		(* Fill input data area with method arguments *)
		MEMSET(ADR(aInputData), 0 ,SIZEOF(aInputData));
		nOffset := 0;
		nOffset := nOffset + MEMCPY(ADR(aInputData)+nOffset, ADR(stMoveToBufferData.stInput),	MIN(SIZEOF(stMoveToBufferData.stInput), (SIZEOF(aInputData)-nOffset)) );
		(* Number of input arguments *)
		nNoOfInputArgs := stMoveToBufferData.iNoOfInputArgs;
		(* Set up input argument information *)
		MEMSET(ADR(aInputArgInfo), 0, SIZEOF(aInputArgInfo));
		aInputArgInfo[1].DataType := eUAType_UInt16;
		aInputArgInfo[1].ValueRank := -1;	// -1: Scalar 
		aInputArgInfo[1].nLenData := SIZEOF(stMoveToBufferData.stInput.eInputType);
		aInputArgInfo[2].DataType := eUAType_String;
		aInputArgInfo[2].ValueRank := -1;	// -1: Scalar 
		aInputArgInfo[2].nLenData := SIZEOF(stMoveToBufferData.stInput.sInput);
		aInputArgInfo[3].DataType := eUAType_String;
		aInputArgInfo[3].ValueRank := -1;	// -1: Scalar 
		aInputArgInfo[3].nLenData := SIZEOF(stMoveToBufferData.stInput.sStationID);
		aInputArgInfo[4].DataType := eUAType_UInt16;
		aInputArgInfo[4].ValueRank := -1;	// -1: Scalar 
		aInputArgInfo[4].nLenData := SIZEOF(stMoveToBufferData.stInput.eStationBufferType);
		aInputArgInfo[5].DataType := eUAType_Byte;
		aInputArgInfo[5].ValueRank := -1;	// -1: Scalar 
		aInputArgInfo[5].nLenData := SIZEOF(stMoveToBufferData.stInput.nIndex);
		aInputArgInfo[6].DataType := eUAType_Byte;
		aInputArgInfo[6].ValueRank := -1;	// -1: Scalar 
		aInputArgInfo[6].nLenData := SIZEOF(stMoveToBufferData.stInput.eDirection);
		aInputArgInfo[7].DataType := eUAType_UInt16;
		aInputArgInfo[7].ValueRank := -1;	// -1: Scalar 
		aInputArgInfo[7].nLenData := SIZEOF(stMoveToBufferData.stInput.nFollowID);
		aInputArgInfo[8].DataType := eUAType_Float;
		aInputArgInfo[8].ValueRank := -1;	// -1: Scalar 
		aInputArgInfo[8].nLenData := SIZEOF(stMoveToBufferData.stInput.fVelocity);
		aInputArgInfo[9].DataType := eUAType_Float;
		aInputArgInfo[9].ValueRank := -1;	// -1: Scalar 
		aInputArgInfo[9].nLenData := SIZEOF(stMoveToBufferData.stInput.fAcceleration);
		
		(* Method outputs *)
		(* Clear output data area *)
		(* Number of output arguments *)
		nNoOfOutputArgs := stMoveToBufferData.iNoOfOutputArgs;
		(* Set up output argument information *)
		MEMSET(ADR(aOutputArgInfo), 0, SIZEOF(aOutputArgInfo));
		aOutputArgInfo[1].DataType := eUAType_Uint16;
		aOutputArgInfo[1].ValueRank := -1;
		aOutputArgInfo[1].nLenData := SIZEOF(stMoveToBufferData.stOutput.eStatus);
		aOutputArgInfo[2].DataType := eUAType_String;
		aOutputArgInfo[2].ValueRank := -1;
		aOutputArgInfo[2].nLenData := SIZEOF(stMoveToBufferData.stOutput.sMessage);
		aOutputArgInfo[3].DataType := eUAType_UInt16;
		aOutputArgInfo[3].ValueRank := -1;
		aOutputArgInfo[3].nLenData := SIZEOF(stMoveToBufferData.stOutput.iCommandID);		
		(* Set up output  *)
		MEMSET(ADR(stMoveToBufferData.stOutput), 0, SIZEOF(stMoveToBufferData.stOutput));
		stMoveToBufferData.stOutput.nNumberOfOutputArguments := nNoOfOutputArgs;
		stMoveToBufferData.stOutput.stOutputArgInfo[1] := aOutputArgInfo[1];
		stMoveToBufferData.stOutput.stOutputArgInfo[2] := aOutputArgInfo[2];
		stMoveToBufferData.stOutput.stOutputArgInfo[3] := aOutputArgInfo[3];
	
		(* Execute FB *)
		fbCallMethod.nNumberOfInputArguments := nNoOfInputArgs;
		fbCallMethod.pInputArgInfo := ADR(aInputArgInfo);
		fbCallMethod.cbInputArgInfo := (SIZEOF(aInputArgInfo[1])*nNoOfInputArgs);
		fbCallMethod.pInputArgData := ADR(aInputData);
		fbCallMethod.cbInputArgData := nOffset;
		fbCallMethod.nNumberOfOutputArguments := nNoOfOutputArgs; 
		fbCallMethod.pOutputArgInfo := ADR(aOutputArgInfo); 
		fbCallMethod.cbOutputArgInfo := (SIZEOF(aOutputArgInfo[1]) * nNoOfOutputArgs); 
		fbCallMethod.pOutputArgInfoAndData := ADR(stMoveToBufferData.stOutput);
		fbCallMethod.cbOutputArgInfoAndData := SIZEOF(stMoveToBufferData.stOutput);
		
		stMoveToBufferData.iStatus := 1;
		bCallMethod := TRUE;
		
	ELSIF ( (stMoveToBufferData.iStatus = 1) AND (stMoveToBufferData.stInput.sInput = sInput) ) THEN
		// Method call Completed...
		IF (eStateMethod = E_TrackClientState.Connected) THEN
			// Method call OK
			IF (stMoveToBufferData.stOutput.eStatus = E_MMServerStatus.eMMServerStatus_Success) THEN
				// Method returned OK
				stMoveToBufferData.iStatus := 2;
				iCmdID := stMoveToBufferData.stOutput.iCommandID;
			ELSE
				// Method returned with error
				stMoveToBufferData.iStatus := 3;
				stMoveToBufferData.stOutput.sMessage;
				iCmdID := 0;
			END_IF
		ELSIF (eStateMethod = E_TrackClientState.Error) THEN
			// Method call failed
			stMoveToBufferData.iStatus := 3;
		END_IF
		
	END_IF
ELSE
	M_CallMoveVehicleToBuffer := -1;
	RETURN;
END_IF

M_CallMoveVehicleToBuffer := stMoveToBufferData.iStatus;
END_METHOD

METHOD M_CallMoveVehicleToDecisionPoint : INT
VAR_INPUT
	eInputType			: E_MMVehicleInputType;
	sInput				: STRING;
	sStationID			: STRING;
	eDirection			: E_MMDirection := E_MMDirection.eMMDirection_Forward;	// Default forward direction
	fVelocity			: REAL;
	fAcceleration		: REAL;
END_VAR
VAR
	i					: UINT;	
END_VAR
VAR_OUTPUT
	iCmdID				: UINT;
END_VAR
IF (stMoveToDecisionPointData.iStatus = 2) OR (stMoveToDecisionPointData.iStatus = 3) THEN
	stMoveToDecisionPointData.iStatus := 0;
END_IF

IF (bConnectedMethod AND NOT bBusyMethod) THEN
	IF (stMoveToDecisionPointData.iStatus = 0) THEN
	(* Setup method calling parameters *)
		(* Method identifier *)
		sObjectIDentifier := stMoveToDecisionPointData.sObjectID;
		sMethodIdentifier := stMoveToDecisionPointData.sMethodID;
	
		(* Method Inputs *)
		stMoveToDecisionPointData.stInput.eInputType := eInputType;
		stMoveToDecisionPointData.stInput.sInput := sInput;
		stMoveToDecisionPointData.stInput.sStationID := sStationID;
		stMoveToDecisionPointData.stInput.eDirection := eDirection;
		stMoveToDecisionPointData.stInput.nFollowID := 0;
		stMoveToDecisionPointData.stInput.fVelocity := fVelocity;
		stMoveToDecisionPointData.stInput.fAcceleration := fAcceleration;
		
		(* Fill input data area with method arguments *)
		MEMSET(ADR(aInputData), 0 ,SIZEOF(aInputData));
		nOffset := 0;
		nOffset := nOffset + MEMCPY(ADR(aInputData)+nOffset, ADR(stMoveToDecisionPointData.stInput),	MIN(SIZEOF(stMoveToDecisionPointData.stInput), (SIZEOF(aInputData)-nOffset)) );
		(* Number of input arguments *)
		nNoOfInputArgs := stMoveToDecisionPointData.iNoOfInputArgs;
		(* Set up input argument information *)
		MEMSET(ADR(aInputArgInfo), 0, SIZEOF(aInputArgInfo));
		aInputArgInfo[1].DataType := eUAType_UInt16;
		aInputArgInfo[1].ValueRank := -1;	// -1: Scalar 
		aInputArgInfo[1].nLenData := SIZEOF(stMoveToDecisionPointData.stInput.eInputType);
		aInputArgInfo[2].DataType := eUAType_String;
		aInputArgInfo[2].ValueRank := -1;	// -1: Scalar 
		aInputArgInfo[2].nLenData := SIZEOF(stMoveToDecisionPointData.stInput.sInput);
		aInputArgInfo[3].DataType := eUAType_String;
		aInputArgInfo[3].ValueRank := -1;	// -1: Scalar 
		aInputArgInfo[3].nLenData := SIZEOF(stMoveToDecisionPointData.stInput.sStationID);
		aInputArgInfo[4].DataType := eUAType_Byte;
		aInputArgInfo[4].ValueRank := -1;	// -1: Scalar 
		aInputArgInfo[4].nLenData := SIZEOF(stMoveToDecisionPointData.stInput.eDirection);
		aInputArgInfo[5].DataType := eUAType_UInt16;
		aInputArgInfo[5].ValueRank := -1;	// -1: Scalar 
		aInputArgInfo[5].nLenData := SIZEOF(stMoveToDecisionPointData.stInput.nFollowID);
		aInputArgInfo[6].DataType := eUAType_Float;
		aInputArgInfo[6].ValueRank := -1;	// -1: Scalar 
		aInputArgInfo[6].nLenData := SIZEOF(stMoveToDecisionPointData.stInput.fVelocity);
		aInputArgInfo[7].DataType := eUAType_Float;
		aInputArgInfo[7].ValueRank := -1;	// -1: Scalar 
		aInputArgInfo[7].nLenData := SIZEOF(stMoveToDecisionPointData.stInput.fAcceleration);
		
		(* Method outputs *)
		(* Clear output data area *)
		(* Number of output arguments *)
		nNoOfOutputArgs := stMoveToDecisionPointData.iNoOfOutputArgs;
		(* Set up output argument information *)
		MEMSET(ADR(aOutputArgInfo), 0, SIZEOF(aOutputArgInfo));
		aOutputArgInfo[1].DataType := eUAType_Uint16;
		aOutputArgInfo[1].ValueRank := -1;
		aOutputArgInfo[1].nLenData := SIZEOF(stMoveToDecisionPointData.stOutput.eStatus);
		aOutputArgInfo[2].DataType := eUAType_String;
		aOutputArgInfo[2].ValueRank := -1;
		aOutputArgInfo[2].nLenData := SIZEOF(stMoveToDecisionPointData.stOutput.sMessage);
		aOutputArgInfo[3].DataType := eUAType_UInt16;
		aOutputArgInfo[3].ValueRank := -1;
		aOutputArgInfo[3].nLenData := SIZEOF(stMoveToDecisionPointData.stOutput.iCommandID);
		(* Set up output  *)
		MEMSET(ADR(stMoveToDecisionPointData.stOutput), 0, SIZEOF(stMoveToDecisionPointData.stOutput));
		stMoveToDecisionPointData.stOutput.nNumberOfOutputArguments := nNoOfOutputArgs;
		stMoveToDecisionPointData.stOutput.stOutputArgInfo[1] := aOutputArgInfo[1];
		stMoveToDecisionPointData.stOutput.stOutputArgInfo[2] := aOutputArgInfo[2];
		stMoveToDecisionPointData.stOutput.stOutputArgInfo[3] := aOutputArgInfo[3];
	
		(* Execute FB *)
		fbCallMethod.nNumberOfInputArguments := nNoOfInputArgs;
		fbCallMethod.pInputArgInfo := ADR(aInputArgInfo);
		fbCallMethod.cbInputArgInfo := (SIZEOF(aInputArgInfo[1])*nNoOfInputArgs);
		fbCallMethod.pInputArgData := ADR(aInputData);
		fbCallMethod.cbInputArgData := nOffset;
		fbCallMethod.nNumberOfOutputArguments := nNoOfOutputArgs; 
		fbCallMethod.pOutputArgInfo := ADR(aOutputArgInfo); 
		fbCallMethod.cbOutputArgInfo := (SIZEOF(aOutputArgInfo[1]) * nNoOfOutputArgs); 
		fbCallMethod.pOutputArgInfoAndData := ADR(stMoveToDecisionPointData.stOutput);
		fbCallMethod.cbOutputArgInfoAndData := SIZEOF(stMoveToDecisionPointData.stOutput);
		
		stMoveToDecisionPointData.iStatus := 1;
		bCallMethod := TRUE;
		
	ELSIF ( (stMoveToDecisionPointData.iStatus = 1) AND (stMoveToDecisionPointData.stInput.sInput = sInput) ) THEN // Make sure it is called from the correct place!
		// Method call Completed...
		IF (eStateMethod = E_TrackClientState.Connected) THEN
			// Method call OK
			IF (stMoveToDecisionPointData.stOutput.eStatus = E_MMServerStatus.eMMServerStatus_Success) THEN
				// Method returned OK
				stMoveToDecisionPointData.iStatus := 2;
				iCmdID := stMoveToDecisionPointData.stOutput.iCommandID;
			ELSE
				// Method returned with error
				stMoveToDecisionPointData.iStatus := 3;
				stMoveToDecisionPointData.stOutput.sMessage;
				iCmdID := 0;
			END_IF
		ELSIF (eStateMethod = E_TrackClientState.Error) THEN
			// Method call failed
			stMoveToDecisionPointData.iStatus := 3;
		END_IF

	END_IF
ELSE
	M_CallMoveVehicleToDecisionPoint := -1;
	RETURN;
END_IF

M_CallMoveVehicleToDecisionPoint := stMoveToDecisionPointData.iStatus;
END_METHOD

METHOD PROTECTED M_CallMoveVehicleToPosition : INT
VAR_INPUT
	eInputType			: E_MMVehicleInputType;
	sInput				: STRING;
	nPathID				: UINT;
	fPosition			: REAL;
	eDirection			: E_MMDirection := E_MMDirection.eMMDirection_Forward;	// Default forward direction
	fVelocity			: REAL;
	fAcceleration		: REAL;
END_VAR
VAR
	i					: UINT;	
END_VAR
VAR_OUTPUT
	iCmdID				: UINT;
END_VAR
IF (stMoveToPositionData.iStatus = 2) OR (stMoveToPositionData.iStatus = 3) THEN
	stMoveToPositionData.iStatus := 0;
END_IF

IF (bConnectedMethod AND NOT bBusyMethod) THEN
	IF (stMoveToPositionData.iStatus = 0) THEN
	(* Setup method calling parameters *)
		(* Method identifier *)
		sObjectIDentifier := stMoveToPositionData.sObjectID;
		sMethodIdentifier := stMoveToPositionData.sMethodID;
	
		(* Method Inputs *)
		stMoveToPositionData.stInput.eInputType := eInputType;
		stMoveToPositionData.stInput.sInput := sInput;
		stMoveToPositionData.stInput.nPathID := nPathID;
		stMoveToPositionData.stInput.fPosition := fPosition;
		stMoveToPositionData.stInput.eDirection := eDirection;
		stMoveToPositionData.stInput.nFollowID := 0;
		stMoveToPositionData.stInput.fVelocity := fVelocity;
		stMoveToPositionData.stInput.fAcceleration := fAcceleration;
		
		(* Fill input data area with method arguments *)
		MEMSET(ADR(aInputData), 0 ,SIZEOF(aInputData));
		nOffset := 0;
		nOffset := nOffset + MEMCPY(ADR(aInputData)+nOffset, ADR(stMoveToPositionData.stInput),	MIN(SIZEOF(stMoveToPositionData.stInput), (SIZEOF(aInputData)-nOffset)) );
		(* Number of input arguments *)
		nNoOfInputArgs := stMoveToPositionData.iNoOfInputArgs;
		(* Set up input argument information *)
		MEMSET(ADR(aInputArgInfo), 0, SIZEOF(aInputArgInfo));
		aInputArgInfo[1].DataType := eUAType_UInt16;
		aInputArgInfo[1].ValueRank := -1;	// -1: Scalar 
		aInputArgInfo[1].nLenData := SIZEOF(stMoveToPositionData.stInput.eInputType);
		aInputArgInfo[2].DataType := eUAType_String;
		aInputArgInfo[2].ValueRank := -1;	// -1: Scalar 
		aInputArgInfo[2].nLenData := SIZEOF(stMoveToPositionData.stInput.sInput);
		aInputArgInfo[3].DataType := eUAType_UInt16;
		aInputArgInfo[3].ValueRank := -1;	// -1: Scalar 
		aInputArgInfo[3].nLenData := SIZEOF(stMoveToPositionData.stInput.nPathID);
		aInputArgInfo[4].DataType := eUAType_Float;
		aInputArgInfo[4].ValueRank := -1;	// -1: Scalar 
		aInputArgInfo[4].nLenData := SIZEOF(stMoveToPositionData.stInput.fPosition);
		aInputArgInfo[5].DataType := eUAType_Byte;
		aInputArgInfo[5].ValueRank := -1;	// -1: Scalar 
		aInputArgInfo[5].nLenData := SIZEOF(stMoveToPositionData.stInput.eDirection);
		aInputArgInfo[6].DataType := eUAType_UInt16;
		aInputArgInfo[6].ValueRank := -1;	// -1: Scalar 
		aInputArgInfo[6].nLenData := SIZEOF(stMoveToPositionData.stInput.nFollowID);
		aInputArgInfo[7].DataType := eUAType_Float;
		aInputArgInfo[7].ValueRank := -1;	// -1: Scalar 
		aInputArgInfo[7].nLenData := SIZEOF(stMoveToPositionData.stInput.fVelocity);
		aInputArgInfo[8].DataType := eUAType_Float;
		aInputArgInfo[8].ValueRank := -1;	// -1: Scalar 
		aInputArgInfo[8].nLenData := SIZEOF(stMoveToPositionData.stInput.fAcceleration);
		
		(* Method outputs *)
		(* Clear output data area *)
		(* Number of output arguments *)
		nNoOfOutputArgs := stMoveToPositionData.iNoOfOutputArgs;
		(* Set up output argument information *)
		MEMSET(ADR(aOutputArgInfo), 0, SIZEOF(aOutputArgInfo));
		aOutputArgInfo[1].DataType := eUAType_Uint16;
		aOutputArgInfo[1].ValueRank := -1;
		aOutputArgInfo[1].nLenData := SIZEOF(stMoveToPositionData.stOutput.eStatus);
		aOutputArgInfo[2].DataType := eUAType_String;
		aOutputArgInfo[2].ValueRank := -1;
		aOutputArgInfo[2].nLenData := SIZEOF(stMoveToPositionData.stOutput.sMessage);
		aOutputArgInfo[3].DataType := eUAType_UInt16;
		aOutputArgInfo[3].ValueRank := -1;
		aOutputArgInfo[3].nLenData := SIZEOF(stMoveToPositionData.stOutput.iCommandID);
		(* Set up output  *)
		MEMSET(ADR(stMoveToPositionData.stOutput), 0, SIZEOF(stMoveToPositionData.stOutput));
		stMoveToPositionData.stOutput.nNumberOfOutputArguments := nNoOfOutputArgs;
		stMoveToPositionData.stOutput.stOutputArgInfo[1] := aOutputArgInfo[1];
		stMoveToPositionData.stOutput.stOutputArgInfo[2] := aOutputArgInfo[2];
		stMoveToPositionData.stOutput.stOutputArgInfo[3] := aOutputArgInfo[3];
	
		(* Execute FB *)
		fbCallMethod.nNumberOfInputArguments := nNoOfInputArgs;
		fbCallMethod.pInputArgInfo := ADR(aInputArgInfo);
		fbCallMethod.cbInputArgInfo := (SIZEOF(aInputArgInfo[1])*nNoOfInputArgs);
		fbCallMethod.pInputArgData := ADR(aInputData);
		fbCallMethod.cbInputArgData := nOffset;
		fbCallMethod.nNumberOfOutputArguments := nNoOfOutputArgs; 
		fbCallMethod.pOutputArgInfo := ADR(aOutputArgInfo); 
		fbCallMethod.cbOutputArgInfo := (SIZEOF(aOutputArgInfo[1]) * nNoOfOutputArgs); 
		fbCallMethod.pOutputArgInfoAndData := ADR(stMoveToPositionData.stOutput);
		fbCallMethod.cbOutputArgInfoAndData := SIZEOF(stMoveToPositionData.stOutput);
		
		stMoveToPositionData.iStatus := 1;
		bCallMethod := TRUE;
		
	ELSIF (stMoveToPositionData.iStatus = 1) THEN
		// Method call Completed...
		IF (sInput = stMoveToPositionData.stInput.sInput) THEN
			// Correct Vehicle identifier ID!
			IF (eStateMethod = E_TrackClientState.Connected) THEN
				// Method call OK
				IF (stMoveToPositionData.stOutput.eStatus = E_MMServerStatus.eMMServerStatus_Success) THEN
					// Method returned OK
					stMoveToPositionData.iStatus := 2;
					iCmdID := stMoveToPositionData.stOutput.iCommandID;
				ELSE
					// Method returned with error
					stMoveToPositionData.iStatus := 3;
					stMoveToPositionData.stOutput.sMessage;
					iCmdId := 0;
				END_IF
			ELSIF (eStateMethod = E_TrackClientState.Error) THEN
				// Method call failed
				stMoveToPositionData.iStatus := 3;
				F_LogLine('TC_MovePos: Method call failed ' , 0);
			END_IF
		
		ELSE
			// Do not allow to return 2 (or 3) if the sInput is not the same as the movment was started with!
			F_LogLine(CONCAT('TC_MovePos: Wrong input: ', sInput) , 0);
			
		END_IF
		
	END_IF
ELSE
	M_CallMoveVehicleToPosition := -1;
	RETURN;
END_IF

M_CallMoveVehicleToPosition := stMoveToPositionData.iStatus;
END_METHOD

METHOD PROTECTED M_CallMoveVehicleToScanner : INT
VAR_INPUT
	eInputType			: E_MMVehicleInputType;
	sInput				: STRING;
	eDirection			: E_MMDirection := E_MMDirection.eMMDirection_Forward;	// Default forward direction
	fVelocity			: REAL;
	fAcceleration		: REAL;
END_VAR
VAR
	i					: UINT;	
	nPostBufferSize: INT;
END_VAR
VAR_OUTPUT
	iCmdID				: UINT;
END_VAR
IF (stMoveToScannerData.iStatus = 2) OR (stMoveToScannerData.iStatus = 3) THEN
	stMoveToScannerData.iStatus := 0;
END_IF

IF (bConnectedMethod AND NOT bBusyMethod) THEN
	IF (stMoveToScannerData.iStatus = 0) THEN
	(* Setup method calling parameters *)
		(* Method identifier *)
		sObjectIDentifier := stMoveToScannerData.sObjectID;
		sMethodIdentifier := stMoveToScannerData.sMethodID;
	
		(* Method Inputs *)
		stMoveToScannerData.stInput.eInputType := eInputType;
		stMoveToScannerData.stInput.sInput := sInput;
		stMoveToScannerData.stInput.eDirection := eDirection;
		stMoveToScannerData.stInput.nFollowID := 0;
		stMoveToScannerData.stInput.fVelocity := fVelocity;
		stMoveToScannerData.stInput.fAcceleration := fAcceleration;
		
		(* Fill input data area with method arguments *)
		MEMSET(ADR(aInputData), 0 ,SIZEOF(aInputData));
		nOffset := 0;
		nOffset := nOffset + MEMCPY(ADR(aInputData)+nOffset, ADR(stMoveToScannerData.stInput),	MIN(SIZEOF(stMoveToScannerData.stInput), (SIZEOF(aInputData)-nOffset)) );
		(* Number of input arguments *)
		nNoOfInputArgs := stMoveToScannerData.iNoOfInputArgs;
		(* Set up input argument information *)
		MEMSET(ADR(aInputArgInfo), 0, SIZEOF(aInputArgInfo));
		aInputArgInfo[1].DataType := eUAType_UInt16;
		aInputArgInfo[1].ValueRank := -1;	// -1: Scalar 
		aInputArgInfo[1].nLenData := SIZEOF(stMoveToScannerData.stInput.eInputType);
		aInputArgInfo[2].DataType := eUAType_String;
		aInputArgInfo[2].ValueRank := -1;	// -1: Scalar 
		aInputArgInfo[2].nLenData := SIZEOF(stMoveToScannerData.stInput.sInput);
		aInputArgInfo[3].DataType := eUAType_Byte;
		aInputArgInfo[3].ValueRank := -1;	// -1: Scalar 
		aInputArgInfo[3].nLenData := SIZEOF(stMoveToScannerData.stInput.eDirection);
		aInputArgInfo[4].DataType := eUAType_UInt16;
		aInputArgInfo[4].ValueRank := -1;	// -1: Scalar 
		aInputArgInfo[4].nLenData := SIZEOF(stMoveToScannerData.stInput.nFollowID);
		aInputArgInfo[5].DataType := eUAType_Float;
		aInputArgInfo[5].ValueRank := -1;	// -1: Scalar 
		aInputArgInfo[5].nLenData := SIZEOF(stMoveToScannerData.stInput.fVelocity);
		aInputArgInfo[6].DataType := eUAType_Float;
		aInputArgInfo[6].ValueRank := -1;	// -1: Scalar 
		aInputArgInfo[6].nLenData := SIZEOF(stMoveToScannerData.stInput.fAcceleration);
		
		(* Method outputs *)
		(* Clear output data area *)
		(* Number of output arguments *)
		nNoOfOutputArgs := stMoveToScannerData.iNoOfOutputArgs;
		(* Set up output argument information *)
		MEMSET(ADR(aOutputArgInfo), 0, SIZEOF(aOutputArgInfo));
		aOutputArgInfo[1].DataType := eUAType_Uint16;
		aOutputArgInfo[1].ValueRank := -1;
		aOutputArgInfo[1].nLenData := SIZEOF(stMoveToScannerData.stOutput.eStatus);
		aOutputArgInfo[2].DataType := eUAType_String;
		aOutputArgInfo[2].ValueRank := -1;
		aOutputArgInfo[2].nLenData := SIZEOF(stMoveToScannerData.stOutput.sMessage);
		aOutputArgInfo[3].DataType := eUAType_UInt16;
		aOutputArgInfo[3].ValueRank := -1;
		aOutputArgInfo[3].nLenData := SIZEOF(stMoveToScannerData.stOutput.iCommandID);
		(* Set up output  *)
		MEMSET(ADR(stMoveToScannerData.stOutput), 0, SIZEOF(stMoveToScannerData.stOutput));
		stMoveToScannerData.stOutput.nNumberOfOutputArguments := nNoOfOutputArgs;
		stMoveToScannerData.stOutput.stOutputArgInfo[1] := aOutputArgInfo[1];
		stMoveToScannerData.stOutput.stOutputArgInfo[2] := aOutputArgInfo[2];
		stMoveToScannerData.stOutput.stOutputArgInfo[3] := aOutputArgInfo[3];
	
		(* Execute FB *)
		fbCallMethod.nNumberOfInputArguments := nNoOfInputArgs;
		fbCallMethod.pInputArgInfo := ADR(aInputArgInfo);
		fbCallMethod.cbInputArgInfo := (SIZEOF(aInputArgInfo[1])*nNoOfInputArgs);
		fbCallMethod.pInputArgData := ADR(aInputData);
		fbCallMethod.cbInputArgData := nOffset;
		fbCallMethod.nNumberOfOutputArguments := nNoOfOutputArgs; 
		fbCallMethod.pOutputArgInfo := ADR(aOutputArgInfo); 
		fbCallMethod.cbOutputArgInfo := (SIZEOF(aOutputArgInfo[1]) * nNoOfOutputArgs); 
		fbCallMethod.pOutputArgInfoAndData := ADR(stMoveToScannerData.stOutput);
		fbCallMethod.cbOutputArgInfoAndData := SIZEOF(stMoveToScannerData.stOutput);
		
		stMoveToScannerData.iStatus := 1;
		bCallMethod := TRUE;
		
	ELSIF (stMoveToScannerData.iStatus = 1) THEN
		// Method call Completed...
		IF (eStateMethod = E_TrackClientState.Connected) THEN
			// Method call OK
			IF (stMoveToScannerData.stOutput.eStatus = E_MMServerStatus.eMMServerStatus_Success) THEN
				// Method returned OK
				stMoveToScannerData.iStatus := 2;
				iCmdID := stMoveToScannerData.stOutput.iCommandID;
			ELSE
				// Method returned with error
				stMoveToScannerData.iStatus := 3;
				stMoveToScannerData.stOutput.sMessage;
				iCmdID := 0;
			END_IF
		ELSIF (eStateMethod = E_TrackClientState.Error) THEN
			// Method call failed
			stMoveToScannerData.iStatus := 3;
		END_IF
		
	END_IF
ELSE
	M_CallMoveVehicleToScanner := -1;
	RETURN;
END_IF

M_CallMoveVehicleToScanner := stMoveToScannerData.iStatus;
END_METHOD

METHOD M_CallMoveVehicleToStationIn : INT
VAR_INPUT
	eInputType			: E_MMVehicleInputType;
	sInput				: STRING;
	sStationID			: STRING;
	eDirection			: E_MMDirection := E_MMDirection.eMMDirection_Forward;	// Default forward direction
	fVelocity			: REAL;
	fAcceleration		: REAL;
END_VAR
VAR
	i					: UINT;	
END_VAR
VAR_OUTPUT
	iCmdID				: UINT;
END_VAR
IF (stMoveToStationInData.iStatus = 2) OR (stMoveToStationInData.iStatus = 3) THEN
	stMoveToStationInData.iStatus := 0;
END_IF

IF (bConnectedMethod AND NOT bBusyMethod) THEN
	IF (stMoveToStationInData.iStatus = 0) THEN
	(* Setup method calling parameters *)
		(* Method identifier *)
		sObjectIDentifier := stMoveToStationInData.sObjectID;
		sMethodIdentifier := stMoveToStationInData.sMethodID;
	
		(* Method Inputs *)
		stMoveToStationInData.stInput.eInputType := eInputType;
		stMoveToStationInData.stInput.sInput := sInput;
		stMoveToStationInData.stInput.sStationID := sStationID;
		stMoveToStationInData.stInput.eDirection := eDirection;
		stMoveToStationInData.stInput.nFollowID := 0;
		stMoveToStationInData.stInput.fVelocity := fVelocity;
		stMoveToStationInData.stInput.fAcceleration := fAcceleration;
		
		(* Fill input data area with method arguments *)
		MEMSET(ADR(aInputData), 0 ,SIZEOF(aInputData));
		nOffset := 0;
		nOffset := nOffset + MEMCPY(ADR(aInputData)+nOffset, ADR(stMoveToStationInData.stInput),	MIN(SIZEOF(stMoveToStationInData.stInput), (SIZEOF(aInputData)-nOffset)) );
		(* Number of input arguments *)
		nNoOfInputArgs := stMoveToStationInData.iNoOfInputArgs;
		(* Set up input argument information *)
		MEMSET(ADR(aInputArgInfo), 0, SIZEOF(aInputArgInfo));
		aInputArgInfo[1].DataType := eUAType_UInt16;
		aInputArgInfo[1].ValueRank := -1;	// -1: Scalar 
		aInputArgInfo[1].nLenData := SIZEOF(stMoveToStationInData.stInput.eInputType);
		aInputArgInfo[2].DataType := eUAType_String;
		aInputArgInfo[2].ValueRank := -1;	// -1: Scalar 
		aInputArgInfo[2].nLenData := SIZEOF(stMoveToStationInData.stInput.sInput);
		aInputArgInfo[3].DataType := eUAType_String;
		aInputArgInfo[3].ValueRank := -1;	// -1: Scalar 
		aInputArgInfo[3].nLenData := SIZEOF(stMoveToStationInData.stInput.sStationID);
		aInputArgInfo[4].DataType := eUAType_Byte;
		aInputArgInfo[4].ValueRank := -1;	// -1: Scalar 
		aInputArgInfo[4].nLenData := SIZEOF(stMoveToStationInData.stInput.eDirection);
		aInputArgInfo[5].DataType := eUAType_UInt16;
		aInputArgInfo[5].ValueRank := -1;	// -1: Scalar 
		aInputArgInfo[5].nLenData := SIZEOF(stMoveToStationInData.stInput.nFollowID);
		aInputArgInfo[6].DataType := eUAType_Float;
		aInputArgInfo[6].ValueRank := -1;	// -1: Scalar 
		aInputArgInfo[6].nLenData := SIZEOF(stMoveToStationInData.stInput.fVelocity);
		aInputArgInfo[7].DataType := eUAType_Float;
		aInputArgInfo[7].ValueRank := -1;	// -1: Scalar 
		aInputArgInfo[7].nLenData := SIZEOF(stMoveToStationInData.stInput.fAcceleration);
		
		(* Method outputs *)
		(* Clear output data area *)
		(* Number of output arguments *)
		nNoOfOutputArgs := stMoveToStationInData.iNoOfOutputArgs;
		(* Set up output argument information *)
		MEMSET(ADR(aOutputArgInfo), 0, SIZEOF(aOutputArgInfo));
		aOutputArgInfo[1].DataType := eUAType_Uint16;
		aOutputArgInfo[1].ValueRank := -1;
		aOutputArgInfo[1].nLenData := SIZEOF(stMoveToStationInData.stOutput.eStatus);
		aOutputArgInfo[2].DataType := eUAType_String;
		aOutputArgInfo[2].ValueRank := -1;
		aOutputArgInfo[2].nLenData := SIZEOF(stMoveToStationInData.stOutput.sMessage);
		aOutputArgInfo[3].DataType := eUAType_UInt16;
		aOutputArgInfo[3].ValueRank := -1;
		aOutputArgInfo[3].nLenData := SIZEOF(stMoveToStationInData.stOutput.iCommandID);
		(* Set up output  *)
		MEMSET(ADR(stMoveToStationInData.stOutput), 0, SIZEOF(stMoveToStationInData.stOutput));
		stMoveToStationInData.stOutput.nNumberOfOutputArguments := nNoOfOutputArgs;
		stMoveToStationInData.stOutput.stOutputArgInfo[1] := aOutputArgInfo[1];
		stMoveToStationInData.stOutput.stOutputArgInfo[2] := aOutputArgInfo[2];
		stMoveToStationInData.stOutput.stOutputArgInfo[3] := aOutputArgInfo[3];
	
		(* Execute FB *)
		fbCallMethod.nNumberOfInputArguments := nNoOfInputArgs;
		fbCallMethod.pInputArgInfo := ADR(aInputArgInfo);
		fbCallMethod.cbInputArgInfo := (SIZEOF(aInputArgInfo[1])*nNoOfInputArgs);
		fbCallMethod.pInputArgData := ADR(aInputData);
		fbCallMethod.cbInputArgData := nOffset;
		fbCallMethod.nNumberOfOutputArguments := nNoOfOutputArgs; 
		fbCallMethod.pOutputArgInfo := ADR(aOutputArgInfo); 
		fbCallMethod.cbOutputArgInfo := (SIZEOF(aOutputArgInfo[1]) * nNoOfOutputArgs); 
		fbCallMethod.pOutputArgInfoAndData := ADR(stMoveToStationInData.stOutput);
		fbCallMethod.cbOutputArgInfoAndData := SIZEOF(stMoveToStationInData.stOutput);
		
		stMoveToStationInData.iStatus := 1;
		bCallMethod := TRUE;
		
	ELSIF ( (stMoveToStationInData.iStatus = 1) AND (stMoveToStationInData.stInput.sInput = sInput) ) THEN
		// Method call Completed...
		IF (eStateMethod = E_TrackClientState.Connected) THEN
			// Method call OK
			IF (stMoveToStationInData.stOutput.eStatus = E_MMServerStatus.eMMServerStatus_Success) THEN
				// Method returned OK
				stMoveToStationInData.iStatus := 2;
				iCmdID := stMoveToStationInData.stOutput.iCommandID;
			ELSE
				// Method returned with error
				stMoveToStationInData.iStatus := 3;
				stMoveToStationInData.stOutput.sMessage;
				iCmdID := 0;
			END_IF
		ELSIF (eStateMethod = E_TrackClientState.Error) THEN
			// Method call failed
			stMoveToStationInData.iStatus := 3;
		END_IF
		
	END_IF
ELSE
	M_CallMoveVehicleToStationIn := -1;
	RETURN;
END_IF

M_CallMoveVehicleToStationIn := stMoveToStationInData.iStatus;
END_METHOD

METHOD PROTECTED M_CallMoveVehicleToStationOut : INT
VAR_INPUT
	eInputType			: E_MMVehicleInputType;
	sInput				: STRING;
	sStationID			: STRING;
	eDirection			: E_MMDirection := E_MMDirection.eMMDirection_Forward;	// Default forward direction
	fVelocity			: REAL;
	fAcceleration		: REAL;
END_VAR
VAR
	i					: UINT;	
	nPostBufferSize: INT;
END_VAR
VAR_OUTPUT
	iCmdID				: UINT;
END_VAR
IF (stMoveToStationOutData.iStatus = 2) OR (stMoveToStationOutData.iStatus = 3) THEN
	stMoveToStationOutData.iStatus := 0;
END_IF

IF (bConnectedMethod AND NOT bBusyMethod) THEN
	IF (stMoveToStationOutData.iStatus = 0) THEN
	(* Setup method calling parameters *)
		(* Method identifier *)
		sObjectIDentifier := stMoveToStationOutData.sObjectID;
		sMethodIdentifier := stMoveToStationOutData.sMethodID;
	
		(* Method Inputs *)
		stMoveToStationOutData.stInput.eInputType := eInputType;
		stMoveToStationOutData.stInput.sInput := sInput;
		stMoveToStationOutData.stInput.sStationID := sStationID;
		stMoveToStationOutData.stInput.eDirection := eDirection;
		stMoveToStationOutData.stInput.nFollowID := 0;
		stMoveToStationOutData.stInput.fVelocity := fVelocity;
		stMoveToStationOutData.stInput.fAcceleration := fAcceleration;
		
		(* Fill input data area with method arguments *)
		MEMSET(ADR(aInputData), 0 ,SIZEOF(aInputData));
		nOffset := 0;
		nOffset := nOffset + MEMCPY(ADR(aInputData)+nOffset, ADR(stMoveToStationOutData.stInput),	MIN(SIZEOF(stMoveToStationOutData.stInput), (SIZEOF(aInputData)-nOffset)) );
		(* Number of input arguments *)
		nNoOfInputArgs := stMoveToStationOutData.iNoOfInputArgs;
		(* Set up input argument information *)
		MEMSET(ADR(aInputArgInfo), 0, SIZEOF(aInputArgInfo));
		aInputArgInfo[1].DataType := eUAType_UInt16;
		aInputArgInfo[1].ValueRank := -1;	// -1: Scalar 
		aInputArgInfo[1].nLenData := SIZEOF(stMoveToStationOutData.stInput.eInputType);
		aInputArgInfo[2].DataType := eUAType_String;
		aInputArgInfo[2].ValueRank := -1;	// -1: Scalar 
		aInputArgInfo[2].nLenData := SIZEOF(stMoveToStationOutData.stInput.sInput);
		aInputArgInfo[3].DataType := eUAType_String;
		aInputArgInfo[3].ValueRank := -1;	// -1: Scalar 
		aInputArgInfo[3].nLenData := SIZEOF(stMoveToStationOutData.stInput.sStationID);
		aInputArgInfo[4].DataType := eUAType_Byte;
		aInputArgInfo[4].ValueRank := -1;	// -1: Scalar 
		aInputArgInfo[4].nLenData := SIZEOF(stMoveToStationOutData.stInput.eDirection);
		aInputArgInfo[5].DataType := eUAType_UInt16;
		aInputArgInfo[5].ValueRank := -1;	// -1: Scalar 
		aInputArgInfo[5].nLenData := SIZEOF(stMoveToStationOutData.stInput.nFollowID);
		aInputArgInfo[6].DataType := eUAType_Float;
		aInputArgInfo[6].ValueRank := -1;	// -1: Scalar 
		aInputArgInfo[6].nLenData := SIZEOF(stMoveToStationOutData.stInput.fVelocity);
		aInputArgInfo[7].DataType := eUAType_Float;
		aInputArgInfo[7].ValueRank := -1;	// -1: Scalar 
		aInputArgInfo[7].nLenData := SIZEOF(stMoveToStationOutData.stInput.fAcceleration);
		
		(* Method outputs *)
		(* Clear output data area *)
		(* Number of output arguments *)
		nNoOfOutputArgs := stMoveToStationOutData.iNoOfOutputArgs;
		(* Set up output argument information *)
		MEMSET(ADR(aOutputArgInfo), 0, SIZEOF(aOutputArgInfo));
		aOutputArgInfo[1].DataType := eUAType_Uint16;
		aOutputArgInfo[1].ValueRank := -1;
		aOutputArgInfo[1].nLenData := SIZEOF(stMoveToStationOutData.stOutput.eStatus);
		aOutputArgInfo[2].DataType := eUAType_String;
		aOutputArgInfo[2].ValueRank := -1;
		aOutputArgInfo[2].nLenData := SIZEOF(stMoveToStationOutData.stOutput.sMessage);
		aOutputArgInfo[3].DataType := eUAType_UInt16;
		aOutputArgInfo[3].ValueRank := -1;
		aOutputArgInfo[3].nLenData := SIZEOF(stMoveToStationOutData.stOutput.iCommandID);
		(* Set up output  *)
		MEMSET(ADR(stMoveToStationOutData.stOutput), 0, SIZEOF(stMoveToStationOutData.stOutput));
		stMoveToStationOutData.stOutput.nNumberOfOutputArguments := nNoOfOutputArgs;
		stMoveToStationOutData.stOutput.stOutputArgInfo[1] := aOutputArgInfo[1];
		stMoveToStationOutData.stOutput.stOutputArgInfo[2] := aOutputArgInfo[2];
		stMoveToStationOutData.stOutput.stOutputArgInfo[3] := aOutputArgInfo[3];
	
		(* Execute FB *)
		fbCallMethod.nNumberOfInputArguments := nNoOfInputArgs;
		fbCallMethod.pInputArgInfo := ADR(aInputArgInfo);
		fbCallMethod.cbInputArgInfo := (SIZEOF(aInputArgInfo[1])*nNoOfInputArgs);
		fbCallMethod.pInputArgData := ADR(aInputData);
		fbCallMethod.cbInputArgData := nOffset;
		fbCallMethod.nNumberOfOutputArguments := nNoOfOutputArgs; 
		fbCallMethod.pOutputArgInfo := ADR(aOutputArgInfo); 
		fbCallMethod.cbOutputArgInfo := (SIZEOF(aOutputArgInfo[1]) * nNoOfOutputArgs); 
		fbCallMethod.pOutputArgInfoAndData := ADR(stMoveToStationOutData.stOutput);
		fbCallMethod.cbOutputArgInfoAndData := SIZEOF(stMoveToStationOutData.stOutput);
		
		stMoveToStationOutData.iStatus := 1;
		bCallMethod := TRUE;
		
	ELSIF ( (stMoveToStationOutData.iStatus = 1) AND (stMoveToStationOutData.stInput.sInput = sInput) ) THEN
		// Method call Completed...
		IF (eStateMethod = E_TrackClientState.Connected) THEN
			// Method call OK
			IF (stMoveToStationOutData.stOutput.eStatus = E_MMServerStatus.eMMServerStatus_Success) THEN
				// Method returned OK
				stMoveToStationOutData.iStatus := 2;
				iCmdID := stMoveToStationOutData.stOutput.iCommandID;
			ELSE
				// Method returned with error
				stMoveToStationOutData.iStatus := 3;
				stMoveToStationOutData.stOutput.sMessage;
				iCmdID := 0;
			END_IF
		ELSIF (eStateMethod = E_TrackClientState.Error) THEN
			// Method call failed
			stMoveToStationOutData.iStatus := 3;
		END_IF
		
	END_IF
ELSE
	M_CallMoveVehicleToStationOut := -1;
	RETURN;
END_IF

M_CallMoveVehicleToStationOut := stMoveToStationOutData.iStatus;
END_METHOD

METHOD PROTECTED M_CallRemovePath : INT
VAR_INPUT
	nPathNo			: UINT;
END_VAR
IF (stRemovePathData.iStatus = 2) OR (stRemovePathData.iStatus = 3) THEN
	stRemovePathData.iStatus := 0;
END_IF

IF (bConnectedMethod AND NOT bBusyMethod) THEN
	IF (stRemovePathData.iStatus = 0) THEN
	(* Setup method calling parameters *)
		(* Method identifier *)
		sObjectIDentifier := stRemovePathData.sObjectID;
		sMethodIdentifier := stRemovePathData.sMethodID;
	
		(* Method Inputs *)
		stRemovePathData.stInput.sCellID := sCellID;
		stRemovePathData.stInput.iPath := nPathNo;
		(* Fill input data area with method arguments *)
		MEMSET(ADR(aInputData), 0 ,SIZEOF(aInputData));
		nOffset := 0;
		nOffset := nOffset + MEMCPY(ADR(aInputData)+nOffset, ADR(stRemovePathData.stInput),	MIN(SIZEOF(stRemovePathData.stInput), (SIZEOF(aInputData)-nOffset)) );
		(* Number of input arguments *)
		nNoOfInputArgs := stRemovePathData.iNoOfInputArgs;
		(* Set up input argument information *)
		MEMSET(ADR(aInputArgInfo), 0, SIZEOF(aInputArgInfo));
		aInputArgInfo[1].DataType := eUAType_String;
		aInputArgInfo[1].ValueRank := -1;	// -1: Scalar 
		aInputArgInfo[1].nLenData := SIZEOF(stRemovePathData.stInput.sCellID);
		aInputArgInfo[2].DataType := eUAType_UInt16;
		aInputArgInfo[2].ValueRank := -1;	// -1: Scalar 
		aInputArgInfo[2].nLenData := SIZEOF(stRemovePathData.stInput.iPath);
		
		(* Method outputs *)
		(* Clear output data area *)
		(* Number of output arguments *)
		nNoOfOutputArgs := stRemovePathData.iNoOfOutputArgs;
		(* Set up output argument information *)
		MEMSET(ADR(aOutputArgInfo), 0, SIZEOF(aOutputArgInfo));
		aOutputArgInfo[1].DataType := eUAType_Uint16;
		aOutputArgInfo[1].ValueRank := -1;
		aOutputArgInfo[1].nLenData := SIZEOF(stRemovePathData.stOutput.eStatus);
		aOutputArgInfo[2].DataType := eUAType_String;
		aOutputArgInfo[2].ValueRank := -1;
		aOutputArgInfo[2].nLenData := SIZEOF(stRemovePathData.stOutput.sMessage);
		(* Set up output  *)
		MEMSET(ADR(stRemovePathData.stOutput), 0, SIZEOF(stRemovePathData.stOutput));
		stRemovePathData.stOutput.nNumberOfOutputArguments := nNoOfOutputArgs;
		stRemovePathData.stOutput.stOutputArgInfo[1] := aOutputArgInfo[1];
		stRemovePathData.stOutput.stOutputArgInfo[2] := aOutputArgInfo[2];
	
		(* Execute FB *)
		fbCallMethod.nNumberOfInputArguments := nNoOfInputArgs;
		fbCallMethod.pInputArgInfo := ADR(aInputArgInfo);
		fbCallMethod.cbInputArgInfo := (SIZEOF(aInputArgInfo[1])*nNoOfInputArgs);
		fbCallMethod.pInputArgData := ADR(aInputData);
		fbCallMethod.cbInputArgData := nOffset;
		fbCallMethod.nNumberOfOutputArguments := nNoOfOutputArgs; 
		fbCallMethod.pOutputArgInfo := ADR(aOutputArgInfo); 
		fbCallMethod.cbOutputArgInfo := (SIZEOF(aOutputArgInfo[1]) * nNoOfOutputArgs); 
		fbCallMethod.pOutputArgInfoAndData := ADR(stRemovePathData.stOutput);
		fbCallMethod.cbOutputArgInfoAndData := SIZEOF(stRemovePathData.stOutput);
		
		stRemovePathData.iStatus := 1;
		bCallMethod := TRUE;
		
	ELSIF (stRemovePathData.iStatus = 1) THEN
		// Method call Completed...
		IF (eStateMethod = E_TrackClientState.Connected) THEN
			// Method call OK
			IF (stRemovePathData.stOutput.eStatus = E_MMServerStatus.eMMServerStatus_Success) THEN
				// Method returned OK
				stRemovePathData.iStatus := 2;
			ELSE
				// Method returned with error
				stRemovePathData.iStatus := 3;
				stRemovePathData.stOutput.sMessage;
			END_IF
		ELSIF (eStateMethod = E_TrackClientState.Error) THEN
			// Method call failed
			stRemovePathData.iStatus := 3;
		END_IF
		
	END_IF
END_IF

M_CallRemovePath := stRemovePathData.iStatus;
END_METHOD

METHOD PROTECTED M_CallRemovePathSegment : INT
VAR_INPUT
	iSegmentNo		: UINT;
END_VAR
IF (stRemovePathSegmentData.iStatus = 2) OR (stRemovePathSegmentData.iStatus = 3) THEN
	stRemovePathSegmentData.iStatus := 0;
END_IF

IF (bConnectedMethod AND NOT bBusyMethod) THEN
	IF (stRemovePathSegmentData.iStatus = 0) THEN
	(* Setup method calling parameters *)
		(* Method identifier *)
		sObjectIDentifier := stRemovePathSegmentData.sObjectID;
		sMethodIdentifier := stRemovePathSegmentData.sMethodID;
	
		(* Method Inputs *)
		stRemovePathSegmentData.stInput.sCellID := sCellID;
		stRemovePathSegmentData.stInput.sSegmentID := CONCAT(sCellID, '_PS');
		stRemovePathSegmentData.stInput.sSegmentID := CONCAT(stRemovePathSegmentData.stInput.sSegmentID, UINT_TO_STRING(iSegmentNo));			
		(* Fill input data area with method arguments *)
		MEMSET(ADR(aInputData), 0 ,SIZEOF(aInputData));
		nOffset := 0;
		nOffset := nOffset + MEMCPY(ADR(aInputData)+nOffset, ADR(stRemovePathSegmentData.stInput),	MIN(SIZEOF(stRemovePathSegmentData.stInput), (SIZEOF(aInputData)-nOffset)) );
		(* Number of input arguments *)
		nNoOfInputArgs := stRemovePathSegmentData.iNoOfInputArgs;
		(* Set up input argument information *)
		MEMSET(ADR(aInputArgInfo), 0, SIZEOF(aInputArgInfo));
		aInputArgInfo[1].DataType := eUAType_String;
		aInputArgInfo[1].ValueRank := -1;	// -1: Scalar 
		aInputArgInfo[1].nLenData := SIZEOF(stRemovePathSegmentData.stInput.sCellID);
		aInputArgInfo[2].DataType := eUAType_String;
		aInputArgInfo[2].ValueRank := -1;	// -1: Scalar 
		aInputArgInfo[2].nLenData := SIZEOF(stRemovePathSegmentData.stInput.sSegmentID);
		
		(* Method outputs *)
		(* Clear output data area *)
		(* Number of output arguments *)
		nNoOfOutputArgs := stRemovePathSegmentData.iNoOfOutputArgs;
		(* Set up output argument information *)
		MEMSET(ADR(aOutputArgInfo), 0, SIZEOF(aOutputArgInfo));
		aOutputArgInfo[1].DataType := eUAType_Uint16;
		aOutputArgInfo[1].ValueRank := -1;
		aOutputArgInfo[1].nLenData := SIZEOF(stRemovePathSegmentData.stOutput.eStatus);
		aOutputArgInfo[2].DataType := eUAType_String;
		aOutputArgInfo[2].ValueRank := -1;
		aOutputArgInfo[2].nLenData := SIZEOF(stRemovePathSegmentData.stOutput.sMessage);
		(* Set up output  *)
		MEMSET(ADR(stRemovePathSegmentData.stOutput), 0, SIZEOF(stRemovePathSegmentData.stOutput));
		stRemovePathSegmentData.stOutput.nNumberOfOutputArguments := nNoOfOutputArgs;
		stRemovePathSegmentData.stOutput.stOutputArgInfo[1] := aOutputArgInfo[1];
		stRemovePathSegmentData.stOutput.stOutputArgInfo[2] := aOutputArgInfo[2];
	
		(* Execute FB *)
		fbCallMethod.nNumberOfInputArguments := nNoOfInputArgs;
		fbCallMethod.pInputArgInfo := ADR(aInputArgInfo);
		fbCallMethod.cbInputArgInfo := (SIZEOF(aInputArgInfo[1])*nNoOfInputArgs);
		fbCallMethod.pInputArgData := ADR(aInputData);
		fbCallMethod.cbInputArgData := nOffset;
		fbCallMethod.nNumberOfOutputArguments := nNoOfOutputArgs; 
		fbCallMethod.pOutputArgInfo := ADR(aOutputArgInfo); 
		fbCallMethod.cbOutputArgInfo := (SIZEOF(aOutputArgInfo[1]) * nNoOfOutputArgs); 
		fbCallMethod.pOutputArgInfoAndData := ADR(stRemovePathSegmentData.stOutput);
		fbCallMethod.cbOutputArgInfoAndData := SIZEOF(stRemovePathSegmentData.stOutput);
		
		stRemovePathSegmentData.iStatus := 1;
		bCallMethod := TRUE;
		
	ELSIF (stRemovePathSegmentData.iStatus = 1) THEN
		// Method call Completed...
		IF (eStateMethod = E_TrackClientState.Connected) THEN
			// Method call OK
			IF (stRemovePathSegmentData.stOutput.eStatus = E_MMServerStatus.eMMServerStatus_Success) THEN
				// Method returned OK
				stRemovePathSegmentData.iStatus := 2;
			ELSE
				// Method returned with error
				stRemovePathSegmentData.iStatus := 3;
				stRemovePathSegmentData.stOutput.sMessage;
			END_IF
		ELSIF (eStateMethod = E_TrackClientState.Error) THEN
			// Method call failed
			stRemovePathSegmentData.iStatus := 3;
		END_IF
		
	END_IF
END_IF

M_CallRemovePathSegment := stRemovePathSegmentData.iStatus;
END_METHOD

METHOD PROTECTED M_CallRemoveReservation : INT
VAR_INPUT
	sStationID					: STRING(30);												(* The identifier for the station. *)
	nTicket						: UINT;														(*  *)
END_VAR
VAR
	i					: UINT;	
END_VAR
IF (stRemoveReservationData.iStatus = 2) OR (stRemoveReservationData.iStatus = 3) THEN
	stRemoveReservationData.iStatus := 0;
END_IF

IF (bConnectedMethod AND NOT bBusyMethod) THEN
	IF (stRemoveReservationData.iStatus = 0) THEN
	(* Setup method calling parameters *)
		(* Method identifier *)
		sObjectIDentifier := stRemoveReservationData.sObjectID;
		sMethodIdentifier := stRemoveReservationData.sMethodID;
	
		(* Method Inputs *)
		stRemoveReservationData.stInput.sStationID := sStationID;
		stRemoveReservationData.stInput.nTicket := nTicket;
		(* Fill input data area with method arguments *)
		MEMSET(ADR(aInputData), 0 ,SIZEOF(aInputData));
		nOffset := 0;
		nOffset := nOffset + MEMCPY(ADR(aInputData)+nOffset, ADR(stRemoveReservationData.stInput),	MIN(SIZEOF(stRemoveReservationData.stInput), (SIZEOF(aInputData)-nOffset)) );
		(* Number of input arguments *)
		nNoOfInputArgs := stRemoveReservationData.iNoOfInputArgs;
		(* Set up input argument information *)
		MEMSET(ADR(aInputArgInfo), 0, SIZEOF(aInputArgInfo));
		aInputArgInfo[1].DataType := eUAType_String;
		aInputArgInfo[1].ValueRank := -1;	// -1: Scalar 
		aInputArgInfo[1].nLenData := SIZEOF(stRemoveReservationData.stInput.sStationID);
		aInputArgInfo[2].DataType := eUAType_UInt16;
		aInputArgInfo[2].ValueRank := -1;	// -1: Scalar 
		aInputArgInfo[2].nLenData := SIZEOF(stRemoveReservationData.stInput.nTicket);
		
		(* Method outputs *)
		(* Clear output data area *)
		(* Number of output arguments *)
		nNoOfOutputArgs := stRemoveReservationData.iNoOfOutputArgs;
		(* Set up output argument information *)
		MEMSET(ADR(aOutputArgInfo), 0, SIZEOF(aOutputArgInfo));
		aOutputArgInfo[1].DataType := eUAType_Uint16;
		aOutputArgInfo[1].ValueRank := -1;
		aOutputArgInfo[1].nLenData := SIZEOF(stRemoveReservationData.stOutput.eStatus);
		aOutputArgInfo[2].DataType := eUAType_String;
		aOutputArgInfo[2].ValueRank := -1;
		aOutputArgInfo[2].nLenData := SIZEOF(stRemoveReservationData.stOutput.sMessage);
		(* Set up output  *)
		MEMSET(ADR(stRemoveReservationData.stOutput), 0, SIZEOF(stRemoveReservationData.stOutput));
		stRemoveReservationData.stOutput.nNumberOfOutputArguments := nNoOfOutputArgs;
		stRemoveReservationData.stOutput.stOutputArgInfo[1] := aOutputArgInfo[1];
		stRemoveReservationData.stOutput.stOutputArgInfo[2] := aOutputArgInfo[2];
	
		(* Execute FB *)
		fbCallMethod.nNumberOfInputArguments := nNoOfInputArgs;
		fbCallMethod.pInputArgInfo := ADR(aInputArgInfo);
		fbCallMethod.cbInputArgInfo := (SIZEOF(aInputArgInfo[1])*nNoOfInputArgs);
		fbCallMethod.pInputArgData := ADR(aInputData);
		fbCallMethod.cbInputArgData := nOffset;
		fbCallMethod.nNumberOfOutputArguments := nNoOfOutputArgs; 
		fbCallMethod.pOutputArgInfo := ADR(aOutputArgInfo); 
		fbCallMethod.cbOutputArgInfo := (SIZEOF(aOutputArgInfo[1]) * nNoOfOutputArgs); 
		fbCallMethod.pOutputArgInfoAndData := ADR(stRemoveReservationData.stOutput);
		fbCallMethod.cbOutputArgInfoAndData := SIZEOF(stRemoveReservationData.stOutput);
		
		stRemoveReservationData.iStatus := 1;
		bCallMethod := TRUE;
		
	ELSIF (stRemoveReservationData.iStatus = 1) THEN
		// Method call Completed...
		IF (eStateMethod = E_TrackClientState.Connected) THEN
			// Method call OK
			IF (stRemoveReservationData.stOutput.eStatus = E_MMServerStatus.eMMServerStatus_Success) THEN
				// Method returned OK
				stRemoveReservationData.iStatus := 2;
			ELSE
				// Method returned with error
				stRemoveReservationData.iStatus := 3;
				stRemoveReservationData.stOutput.sMessage;
			END_IF
		ELSIF (eStateMethod = E_TrackClientState.Error) THEN
			// Method call failed
			stRemoveReservationData.iStatus := 3;
		END_IF
		
	END_IF
END_IF

M_CallRemoveReservation := stRemoveReservationData.iStatus;
END_METHOD

METHOD PROTECTED M_CallRemoveStation : INT
VAR_INPUT
	nStationNo			: UINT(1..5);
END_VAR
IF (stRemoveStationData.iStatus = 2) OR (stRemoveStationData.iStatus = 3) THEN
	stRemoveStationData.iStatus := 0;
END_IF

IF (bConnectedMethod AND NOT bBusyMethod) THEN
	IF (stRemoveStationData.iStatus = 0) THEN
	(* Setup method calling parameters *)
		(* Method identifier *)
		sObjectIDentifier := stRemoveStationData.sObjectID;
		sMethodIdentifier := stRemoveStationData.sMethodID;
	
		(* Method Inputs *)
		stRemoveStationData.stInput.sCellID := sCellID;
		stRemoveStationData.stInput.sStationID := aStations[nStationNo].sStationID;
		(* Fill input data area with method arguments *)
		MEMSET(ADR(aInputData), 0 ,SIZEOF(aInputData));
		nOffset := 0;
		nOffset := nOffset + MEMCPY(ADR(aInputData)+nOffset, ADR(stRemoveStationData.stInput),	MIN(SIZEOF(stRemoveStationData.stInput), (SIZEOF(aInputData)-nOffset)) );
		(* Number of input arguments *)
		nNoOfInputArgs := stRemoveStationData.iNoOfInputArgs;
		(* Set up input argument information *)
		MEMSET(ADR(aInputArgInfo), 0, SIZEOF(aInputArgInfo));
		aInputArgInfo[1].DataType := eUAType_String;
		aInputArgInfo[1].ValueRank := -1;	// -1: Scalar 
		aInputArgInfo[1].nLenData := SIZEOF(stRemoveStationData.stInput.sCellID);
		aInputArgInfo[2].DataType := eUAType_String;
		aInputArgInfo[2].ValueRank := -1;	// -1: Scalar 
		aInputArgInfo[2].nLenData := SIZEOF(stRemoveStationData.stInput.sStationID);
		
		(* Method outputs *)
		(* Clear output data area *)
		(* Number of output arguments *)
		nNoOfOutputArgs := stRemoveStationData.iNoOfOutputArgs;
		(* Set up output argument information *)
		MEMSET(ADR(aOutputArgInfo), 0, SIZEOF(aOutputArgInfo));
		aOutputArgInfo[1].DataType := eUAType_Uint16;
		aOutputArgInfo[1].ValueRank := -1;
		aOutputArgInfo[1].nLenData := SIZEOF(stRemoveStationData.stOutput.eStatus);
		aOutputArgInfo[2].DataType := eUAType_String;
		aOutputArgInfo[2].ValueRank := -1;
		aOutputArgInfo[2].nLenData := SIZEOF(stRemoveStationData.stOutput.sMessage);
		(* Set up output  *)
		MEMSET(ADR(stRemoveStationData.stOutput), 0, SIZEOF(stRemoveStationData.stOutput));
		stRemoveStationData.stOutput.nNumberOfOutputArguments := nNoOfOutputArgs;
		stRemoveStationData.stOutput.stOutputArgInfo[1] := aOutputArgInfo[1];
		stRemoveStationData.stOutput.stOutputArgInfo[2] := aOutputArgInfo[2];
	
		(* Execute FB *)
		fbCallMethod.nNumberOfInputArguments := nNoOfInputArgs;
		fbCallMethod.pInputArgInfo := ADR(aInputArgInfo);
		fbCallMethod.cbInputArgInfo := (SIZEOF(aInputArgInfo[1])*nNoOfInputArgs);
		fbCallMethod.pInputArgData := ADR(aInputData);
		fbCallMethod.cbInputArgData := nOffset;
		fbCallMethod.nNumberOfOutputArguments := nNoOfOutputArgs; 
		fbCallMethod.pOutputArgInfo := ADR(aOutputArgInfo); 
		fbCallMethod.cbOutputArgInfo := (SIZEOF(aOutputArgInfo[1]) * nNoOfOutputArgs); 
		fbCallMethod.pOutputArgInfoAndData := ADR(stRemoveStationData.stOutput);
		fbCallMethod.cbOutputArgInfoAndData := SIZEOF(stRemoveStationData.stOutput);
		
		stRemoveStationData.iStatus := 1;
		bCallMethod := TRUE;
		
	ELSIF (stRemoveStationData.iStatus = 1) THEN
		// Method call Completed...
		IF (eStateMethod = E_TrackClientState.Connected) THEN
			// Method call OK
			IF (stRemoveStationData.stOutput.eStatus = E_MMServerStatus.eMMServerStatus_Success) THEN
				// Method returned OK
				stRemoveStationData.iStatus := 2;
			ELSE
				// Method returned with error
				stRemoveStationData.iStatus := 3;
				stRemoveStationData.stOutput.sMessage;
			END_IF
		ELSIF (eStateMethod = E_TrackClientState.Error) THEN
			// Method call failed
			stRemoveStationData.iStatus := 3;
		END_IF
		
	END_IF
END_IF

M_CallRemoveStation := stRemoveStationData.iStatus;
END_METHOD

METHOD PROTECTED M_CallRemoveTrafficLight : INT
VAR_INPUT
END_VAR
IF (stRemoveTrafficLightData.iStatus = 2) OR (stRemoveTrafficLightData.iStatus = 3) THEN
	stRemoveTrafficLightData.iStatus := 0;
END_IF

IF (bConnectedMethod AND NOT bBusyMethod) THEN
	IF (stRemoveTrafficLightData.iStatus = 0) THEN
	(* Setup method calling parameters *)
		(* Method identifier *)
		sObjectIDentifier := stRemoveTrafficLightData.sObjectID;
		sMethodIdentifier := stRemoveTrafficLightData.sMethodID;
	
		(* Method Inputs *)
		stRemoveTrafficLightData.stInput.sCellID := sCellID;
		stRemoveTrafficLightData.stInput.sID := CONCAT(sCellID, '_TL');
		(* Fill input data area with method arguments *)
		MEMSET(ADR(aInputData), 0 ,SIZEOF(aInputData));
		nOffset := 0;
		nOffset := nOffset + MEMCPY(ADR(aInputData)+nOffset, ADR(stRemoveTrafficLightData.stInput),	MIN(SIZEOF(stRemoveTrafficLightData.stInput),	(SIZEOF(aInputData)-nOffset)) );
		(* Number of input arguments *)
		nNoOfInputArgs := stRemoveTrafficLightData.iNoOfInputArgs;
		(* Set up input argument information *)
		MEMSET(ADR(aInputArgInfo), 0, SIZEOF(aInputArgInfo));
		aInputArgInfo[1].DataType := eUAType_String;
		aInputArgInfo[1].ValueRank := -1;	// -1: Scalar 
		aInputArgInfo[1].nLenData := SIZEOF(stRemoveTrafficLightData.stInput.sCellID);
		aInputArgInfo[2].DataType := eUAType_String;
		aInputArgInfo[2].ValueRank := -1;	// -1: Scalar 
		aInputArgInfo[2].nLenData := SIZEOF(stRemoveTrafficLightData.stInput.sID);
		
		(* Method outputs *)
		(* Clear output data area *)
		(* Number of output arguments *)
		nNoOfOutputArgs := stRemoveTrafficLightData.iNoOfOutputArgs;
		(* Set up output argument information *)
		MEMSET(ADR(aOutputArgInfo), 0, SIZEOF(aOutputArgInfo));
		aOutputArgInfo[1].DataType := eUAType_Uint16;
		aOutputArgInfo[1].ValueRank := -1;
		aOutputArgInfo[1].nLenData := SIZEOF(stRemoveTrafficLightData.stOutput.eStatus);
		aOutputArgInfo[2].DataType := eUAType_String;
		aOutputArgInfo[2].ValueRank := -1;
		aOutputArgInfo[2].nLenData := SIZEOF(stRemoveTrafficLightData.stOutput.sMessage);
		(* Set up output  *)
		MEMSET(ADR(stRemoveTrafficLightData.stOutput), 0, SIZEOF(stRemoveTrafficLightData.stOutput));
		stRemoveTrafficLightData.stOutput.nNumberOfOutputArguments := nNoOfOutputArgs;
		stRemoveTrafficLightData.stOutput.stOutputArgInfo[1] := aOutputArgInfo[1];
		stRemoveTrafficLightData.stOutput.stOutputArgInfo[2] := aOutputArgInfo[2];
	
		(* Execute FB *)
		fbCallMethod.nNumberOfInputArguments := nNoOfInputArgs;
		fbCallMethod.pInputArgInfo := ADR(aInputArgInfo);
		fbCallMethod.cbInputArgInfo := (SIZEOF(aInputArgInfo[1])*nNoOfInputArgs);
		fbCallMethod.pInputArgData := ADR(aInputData);
		fbCallMethod.cbInputArgData := nOffset;
		fbCallMethod.nNumberOfOutputArguments := nNoOfOutputArgs; 
		fbCallMethod.pOutputArgInfo := ADR(aOutputArgInfo); 
		fbCallMethod.cbOutputArgInfo := (SIZEOF(aOutputArgInfo[1]) * nNoOfOutputArgs); 
		fbCallMethod.pOutputArgInfoAndData := ADR(stRemoveTrafficLightData.stOutput);
		fbCallMethod.cbOutputArgInfoAndData := SIZEOF(stRemoveTrafficLightData.stOutput);
		
		stRemoveTrafficLightData.iStatus := 1;
		bCallMethod := TRUE;
		
	ELSIF (stRemoveTrafficLightData.iStatus = 1) THEN
		// Method call Completed...
		IF (eStateMethod = E_TrackClientState.Connected) THEN
			// Method call OK
			IF (stRemoveTrafficLightData.stOutput.eStatus = E_MMServerStatus.eMMServerStatus_Success) THEN
				// Method returned OK
				stRemoveTrafficLightData.iStatus := 2;
			ELSE
				// Method returned with error
				stRemoveTrafficLightData.iStatus := 3;
				stRemoveTrafficLightData.stOutput.sMessage;
			END_IF
		ELSIF (eStateMethod = E_TrackClientState.Error) THEN
			// Method call failed
			stRemoveTrafficLightData.iStatus := 3;
		END_IF
		
	END_IF
END_IF

M_CallRemoveTrafficLight := stRemoveTrafficLightData.iStatus;
END_METHOD

METHOD PROTECTED M_CallResetPath : INT
VAR_INPUT
	nPathNo			: UINT(1..5);
END_VAR
IF (stResetPathData.iStatus = 2) OR (stResetPathData.iStatus = 3) THEN
	stResetPathData.iStatus := 0;
END_IF

IF (bConnectedMethod AND NOT bBusyMethod) THEN
	IF (stResetPathData.iStatus = 0) THEN
	(* Setup method calling parameters *)
		(* Method identifier *)
		sObjectIDentifier := stResetPathData.sObjectID;
		sMethodIdentifier := stResetPathData.sMethodID;
	
		(* Method Inputs *)
		stResetPathData.stInput.iPath := nPathNo;
		(* Fill input data area with method arguments *)
		MEMSET(ADR(aInputData), 0 ,SIZEOF(aInputData));
		nOffset := 0;
		nOffset := nOffset + MEMCPY(ADR(aInputData)+nOffset, ADR(stResetPathData.stInput),	MIN(SIZEOF(stResetPathData.stInput), (SIZEOF(aInputData)-nOffset)) );
		(* Number of input arguments *)
		nNoOfInputArgs := stResetPathData.iNoOfInputArgs;
		(* Set up input argument information *)
		MEMSET(ADR(aInputArgInfo), 0, SIZEOF(aInputArgInfo));
		aInputArgInfo[1].DataType := eUAType_UInt16;
		aInputArgInfo[1].ValueRank := -1;	// -1: Scalar 
		aInputArgInfo[1].nLenData := SIZEOF(stResetPathData.stInput.iPath);
		
		(* Method outputs *)
		(* Clear output data area *)
		(* Number of output arguments *)
		nNoOfOutputArgs := stResetPathData.iNoOfOutputArgs;
		(* Set up output argument information *)
		MEMSET(ADR(aOutputArgInfo), 0, SIZEOF(aOutputArgInfo));
		aOutputArgInfo[1].DataType := eUAType_Uint16;
		aOutputArgInfo[1].ValueRank := -1;
		aOutputArgInfo[1].nLenData := SIZEOF(stResetPathData.stOutput.eStatus);
		aOutputArgInfo[2].DataType := eUAType_String;
		aOutputArgInfo[2].ValueRank := -1;
		aOutputArgInfo[2].nLenData := SIZEOF(stResetPathData.stOutput.sMessage);
		(* Set up output  *)
		MEMSET(ADR(stResetPathData.stOutput), 0, SIZEOF(stResetPathData.stOutput));
		stResetPathData.stOutput.nNumberOfOutputArguments := nNoOfOutputArgs;
		stResetPathData.stOutput.stOutputArgInfo[1] := aOutputArgInfo[1];
		stResetPathData.stOutput.stOutputArgInfo[2] := aOutputArgInfo[2];
	
		(* Execute FB *)
		fbCallMethod.nNumberOfInputArguments := nNoOfInputArgs;
		fbCallMethod.pInputArgInfo := ADR(aInputArgInfo);
		fbCallMethod.cbInputArgInfo := (SIZEOF(aInputArgInfo[1])*nNoOfInputArgs);
		fbCallMethod.pInputArgData := ADR(aInputData);
		fbCallMethod.cbInputArgData := nOffset;
		fbCallMethod.nNumberOfOutputArguments := nNoOfOutputArgs; 
		fbCallMethod.pOutputArgInfo := ADR(aOutputArgInfo); 
		fbCallMethod.cbOutputArgInfo := (SIZEOF(aOutputArgInfo[1]) * nNoOfOutputArgs); 
		fbCallMethod.pOutputArgInfoAndData := ADR(stResetPathData.stOutput);
		fbCallMethod.cbOutputArgInfoAndData := SIZEOF(stResetPathData.stOutput);
		
		stResetPathData.iStatus := 1;
		bCallMethod := TRUE;
		
	ELSIF (stResetPathData.iStatus = 1) THEN
		// Method call Completed...
		IF (eStateMethod = E_TrackClientState.Connected) THEN
			// eStateMethod call OK
			IF (stResetPathData.stOutput.eStatus = E_MMServerStatus.eMMServerStatus_Success) THEN
				// Method returned OK
				stResetPathData.iStatus := 2;
			ELSE
				// Method returned with error
				stResetPathData.iStatus := 3;
				stResetPathData.stOutput.sMessage;
			END_IF
		ELSIF (eStateMethod = E_TrackClientState.Error) THEN
			// Method call failed
			stResetPathData.iStatus := 3;
		END_IF
		
	END_IF
END_IF

M_CallResetPath := stResetPathData.iStatus;
END_METHOD

METHOD PROTECTED M_CallResumePath : INT
VAR_INPUT
	nPathNo			: UINT(1..5);
END_VAR
IF (stResumePathData.iStatus = 2) OR (stResumePathData.iStatus = 3) THEN
	stResumePathData.iStatus := 0;
END_IF

IF (bConnectedMethod AND NOT bBusyMethod) THEN
	IF (stResumePathData.iStatus = 0) THEN
	(* Setup method calling parameters *)
		(* Method identifier *)
		sObjectIDentifier := stResumePathData.sObjectID;
		sMethodIdentifier := stResumePathData.sMethodID;
	
		(* Method Inputs *)
		stResumePathData.stInput.iPath := nPathNo;
		(* Fill input data area with method arguments *)
		MEMSET(ADR(aInputData), 0 ,SIZEOF(aInputData));
		nOffset := 0;
		nOffset := nOffset + MEMCPY(ADR(aInputData)+nOffset, ADR(stResumePathData.stInput),	MIN(SIZEOF(stResumePathData.stInput), (SIZEOF(aInputData)-nOffset)) );
		(* Number of input arguments *)
		nNoOfInputArgs := stResumePathData.iNoOfInputArgs;
		(* Set up input argument information *)
		MEMSET(ADR(aInputArgInfo), 0, SIZEOF(aInputArgInfo));
		aInputArgInfo[1].DataType := eUAType_UInt16;
		aInputArgInfo[1].ValueRank := -1;	// -1: Scalar 
		aInputArgInfo[1].nLenData := SIZEOF(stResumePathData.stInput.iPath);
		
		(* Method outputs *)
		(* Clear output data area *)
		(* Number of output arguments *)
		nNoOfOutputArgs := stResumePathData.iNoOfOutputArgs;
		(* Set up output argument information *)
		MEMSET(ADR(aOutputArgInfo), 0, SIZEOF(aOutputArgInfo));
		aOutputArgInfo[1].DataType := eUAType_Uint16;
		aOutputArgInfo[1].ValueRank := -1;
		aOutputArgInfo[1].nLenData := SIZEOF(stResumePathData.stOutput.eStatus);
		aOutputArgInfo[2].DataType := eUAType_String;
		aOutputArgInfo[2].ValueRank := -1;
		aOutputArgInfo[2].nLenData := SIZEOF(stResumePathData.stOutput.sMessage);
		(* Set up output  *)
		MEMSET(ADR(stResumePathData.stOutput), 0, SIZEOF(stResumePathData.stOutput));
		stResumePathData.stOutput.nNumberOfOutputArguments := nNoOfOutputArgs;
		stResumePathData.stOutput.stOutputArgInfo[1] := aOutputArgInfo[1];
		stResumePathData.stOutput.stOutputArgInfo[2] := aOutputArgInfo[2];
	
		(* Execute FB *)
		fbCallMethod.nNumberOfInputArguments := nNoOfInputArgs;
		fbCallMethod.pInputArgInfo := ADR(aInputArgInfo);
		fbCallMethod.cbInputArgInfo := (SIZEOF(aInputArgInfo[1])*nNoOfInputArgs);
		fbCallMethod.pInputArgData := ADR(aInputData);
		fbCallMethod.cbInputArgData := nOffset;
		fbCallMethod.nNumberOfOutputArguments := nNoOfOutputArgs; 
		fbCallMethod.pOutputArgInfo := ADR(aOutputArgInfo); 
		fbCallMethod.cbOutputArgInfo := (SIZEOF(aOutputArgInfo[1]) * nNoOfOutputArgs); 
		fbCallMethod.pOutputArgInfoAndData := ADR(stResumePathData.stOutput);
		fbCallMethod.cbOutputArgInfoAndData := SIZEOF(stResumePathData.stOutput);
		
		stResumePathData.iStatus := 1;
		bCallMethod := TRUE;
		
	ELSIF (stResumePathData.iStatus = 1) THEN
		// Method call Completed...
		IF (eStateMethod = E_TrackClientState.Connected) THEN
			// Method call OK
			IF (stResumePathData.stOutput.eStatus = E_MMServerStatus.eMMServerStatus_Success) THEN
				// Method returned OK
				stResumePathData.iStatus := 2;
			ELSE
				// Method returned with error
				stResumePathData.iStatus := 3;
				stResumePathData.stOutput.sMessage;
			END_IF
		ELSIF (eStateMethod = E_TrackClientState.Error) THEN
			// Method call failed
			stResumePathData.iStatus := 3;
		END_IF
		
	END_IF
END_IF

M_CallResumePath := stResumePathData.iStatus;
END_METHOD

METHOD PROTECTED M_CallSetTrafficLightColor : INT
VAR_INPUT
	nTrafficLightNo	: UINT;
	nColor			: INT;
END_VAR
IF (stSetTrafficLightColorData.iStatus = 2) OR (stSetTrafficLightColorData.iStatus = 3) THEN
	stSetTrafficLightColorData.iStatus := 0;
END_IF

IF (bConnectedMethod AND NOT bBusyMethod) THEN
	IF (stSetTrafficLightColorData.iStatus = 0) THEN
	(* Setup method calling parameters *)
		(* Method identifier *)
		sObjectIDentifier := stSetTrafficLightColorData.sObjectID;
		sMethodIdentifier := stSetTrafficLightColorData.sMethodID;
			
		(* Method Inputs *)
		stSetTrafficLightColorData.stInput.sCellID := sCellID;
		stSetTrafficLightColorData.stInput.sID := CONCAT(sCellID, '_TL');
		stSetTrafficLightColorData.stInput.sID := CONCAT(stSetTrafficLightColorData.stInput.sID, UINT_TO_STRING(nTrafficLightNo));
		stSetTrafficLightColorData.stInput.nColor := nColor;
		(* Fill input data area with method arguments *)
		MEMSET(ADR(aInputData), 0 ,SIZEOF(aInputData));
		nOffset := 0;
		nOffset := nOffset + MEMCPY(ADR(aInputData)+nOffset, ADR(stSetTrafficLightColorData.stInput),	MIN(SIZEOF(stSetTrafficLightColorData.stInput),	(SIZEOF(aInputData)-nOffset)) );
		(* Number of input arguments *)
		nNoOfInputArgs := stSetTrafficLightColorData.iNoOfInputArgs;
		(* Set up input argument information *)
		MEMSET(ADR(aInputArgInfo), 0, SIZEOF(aInputArgInfo));
		aInputArgInfo[1].DataType := eUAType_String;
		aInputArgInfo[1].ValueRank := -1;	// -1: Scalar 
		aInputArgInfo[1].nLenData := SIZEOF(stSetTrafficLightColorData.stInput.sCellID);
		aInputArgInfo[2].DataType := eUAType_String;
		aInputArgInfo[2].ValueRank := -1;	// -1: Scalar 
		aInputArgInfo[2].nLenData := SIZEOF(stSetTrafficLightColorData.stInput.sID);
		aInputArgInfo[3].DataType := eUAType_Int16;
		aInputArgInfo[3].ValueRank := -1;	// -1: Scalar 
		aInputArgInfo[3].nLenData := SIZEOF(nColor);
		
		(* Method outputs *)
		(* Clear output data area *)
		(* Number of output arguments *)
		nNoOfOutputArgs := stSetTrafficLightColorData.iNoOfOutputArgs;
		(* Set up output argument information *)
		MEMSET(ADR(aOutputArgInfo), 0, SIZEOF(aOutputArgInfo));
		aOutputArgInfo[1].DataType := eUAType_Uint16;
		aOutputArgInfo[1].ValueRank := -1;
		aOutputArgInfo[1].nLenData := SIZEOF(stSetTrafficLightColorData.stOutput.eStatus);
		aOutputArgInfo[2].DataType := eUAType_String;
		aOutputArgInfo[2].ValueRank := -1;
		aOutputArgInfo[2].nLenData := SIZEOF(stSetTrafficLightColorData.stOutput.sMessage);
		(* Set up output  *)
		MEMSET(ADR(stSetTrafficLightColorData.stOutput), 0, SIZEOF(stSetTrafficLightColorData.stOutput));
		stSetTrafficLightColorData.stOutput.nNumberOfOutputArguments := nNoOfOutputArgs;
		stSetTrafficLightColorData.stOutput.stOutputArgInfo[1] := aOutputArgInfo[1];
		stSetTrafficLightColorData.stOutput.stOutputArgInfo[2] := aOutputArgInfo[2];
	
		(* Execute FB *)
		fbCallMethod.nNumberOfInputArguments := nNoOfInputArgs;
		fbCallMethod.pInputArgInfo := ADR(aInputArgInfo);
		fbCallMethod.cbInputArgInfo := (SIZEOF(aInputArgInfo[1])*nNoOfInputArgs);
		fbCallMethod.pInputArgData := ADR(aInputData);
		fbCallMethod.cbInputArgData := nOffset;
		fbCallMethod.nNumberOfOutputArguments := nNoOfOutputArgs; 
		fbCallMethod.pOutputArgInfo := ADR(aOutputArgInfo); 
		fbCallMethod.cbOutputArgInfo := (SIZEOF(aOutputArgInfo[1]) * nNoOfOutputArgs); 
		fbCallMethod.pOutputArgInfoAndData := ADR(stSetTrafficLightColorData.stOutput);
		fbCallMethod.cbOutputArgInfoAndData := SIZEOF(stSetTrafficLightColorData.stOutput);
		
		stSetTrafficLightColorData.iStatus := 1;
		bCallMethod := TRUE;
		
	ELSIF (stSetTrafficLightColorData.iStatus = 1) THEN
		// Method call Completed...
		IF (eStateMethod = E_TrackClientState.Connected) THEN
			// Method call OK
			IF (stSetTrafficLightColorData.stOutput.eStatus = E_MMServerStatus.eMMServerStatus_Success) THEN
				// Method returned OK
				stSetTrafficLightColorData.iStatus := 2;
			ELSE
				// Method returned with error
				stSetTrafficLightColorData.iStatus := 3;
				stSetTrafficLightColorData.stOutput.sMessage;
			END_IF
		ELSIF (eStateMethod = E_TrackClientState.Error) THEN
			// Method call failed
			stSetTrafficLightColorData.iStatus := 3;
		END_IF
		
	END_IF
END_IF

M_CallSetTrafficLightColor := stSetTrafficLightColorData.iStatus;
END_METHOD

METHOD PROTECTED M_CallStartPath : INT
VAR_INPUT
	nPathNo			: UINT(1..5);
END_VAR
IF (stStartPathData.iStatus = 2) OR (stStartPathData.iStatus = 3) THEN
	stStartPathData.iStatus := 0;
END_IF

IF (bConnectedMethod AND NOT bBusyMethod) THEN
	IF (stStartPathData.iStatus = 0) THEN
	(* Setup method calling parameters *)
		(* Method identifier *)
		sObjectIDentifier := stStartPathData.sObjectID;
		sMethodIdentifier := stStartPathData.sMethodID;
	
		(* Method Inputs *)
		stStartPathData.stInput.iPath := nPathNo;
		(* Fill input data area with method arguments *)
		MEMSET(ADR(aInputData), 0 ,SIZEOF(aInputData));
		nOffset := 0;
		nOffset := nOffset + MEMCPY(ADR(aInputData)+nOffset, ADR(stStartPathData.stInput),	MIN(SIZEOF(stStartPathData.stInput), (SIZEOF(aInputData)-nOffset)) );
		(* Number of input arguments *)
		nNoOfInputArgs := stStartPathData.iNoOfInputArgs;
		(* Set up input argument information *)
		MEMSET(ADR(aInputArgInfo), 0, SIZEOF(aInputArgInfo));
		aInputArgInfo[1].DataType := eUAType_UInt16;
		aInputArgInfo[1].ValueRank := -1;	// -1: Scalar 
		aInputArgInfo[1].nLenData := SIZEOF(stStartPathData.stInput.iPath);
		
		(* Method outputs *)
		(* Clear output data area *)
		(* Number of output arguments *)
		nNoOfOutputArgs := stStartPathData.iNoOfOutputArgs;
		(* Set up output argument information *)
		MEMSET(ADR(aOutputArgInfo), 0, SIZEOF(aOutputArgInfo));
		aOutputArgInfo[1].DataType := eUAType_Uint16;
		aOutputArgInfo[1].ValueRank := -1;
		aOutputArgInfo[1].nLenData := SIZEOF(stStartPathData.stOutput.eStatus);
		aOutputArgInfo[2].DataType := eUAType_String;
		aOutputArgInfo[2].ValueRank := -1;
		aOutputArgInfo[2].nLenData := SIZEOF(stStartPathData.stOutput.sMessage);
		(* Set up output  *)
		MEMSET(ADR(stStartPathData.stOutput), 0, SIZEOF(stStartPathData.stOutput));
		stStartPathData.stOutput.nNumberOfOutputArguments := nNoOfOutputArgs;
		stStartPathData.stOutput.stOutputArgInfo[1] := aOutputArgInfo[1];
		stStartPathData.stOutput.stOutputArgInfo[2] := aOutputArgInfo[2];
	
		(* Execute FB *)
		fbCallMethod.nNumberOfInputArguments := nNoOfInputArgs;
		fbCallMethod.pInputArgInfo := ADR(aInputArgInfo);
		fbCallMethod.cbInputArgInfo := (SIZEOF(aInputArgInfo[1])*nNoOfInputArgs);
		fbCallMethod.pInputArgData := ADR(aInputData);
		fbCallMethod.cbInputArgData := nOffset;
		fbCallMethod.nNumberOfOutputArguments := nNoOfOutputArgs; 
		fbCallMethod.pOutputArgInfo := ADR(aOutputArgInfo); 
		fbCallMethod.cbOutputArgInfo := (SIZEOF(aOutputArgInfo[1]) * nNoOfOutputArgs); 
		fbCallMethod.pOutputArgInfoAndData := ADR(stStartPathData.stOutput);
		fbCallMethod.cbOutputArgInfoAndData := SIZEOF(stStartPathData.stOutput);
		
		stStartPathData.iStatus := 1;
		bCallMethod := TRUE;
		
	ELSIF (stStartPathData.iStatus = 1) THEN
		// Method call Completed...
		IF (eStateMethod = E_TrackClientState.Connected) THEN
			// Method call OK
			IF (stStartPathData.stOutput.eStatus = E_MMServerStatus.eMMServerStatus_Success) THEN
				// Method returned OK
				stStartPathData.iStatus := 2;
			ELSE
				// Method returned with error
				stStartPathData.iStatus := 3;
				stStartPathData.stOutput.sMessage;
			END_IF
		ELSIF (eStateMethod = E_TrackClientState.Error) THEN
			// Method call failed
			stStartPathData.iStatus := 3;
		END_IF
		
	END_IF
END_IF

M_CallStartPath := stStartPathData.iStatus;
END_METHOD

METHOD PROTECTED M_CallSuspendPath : INT
VAR_INPUT
	nPathNo			: UINT(1..5);
END_VAR
IF (stSuspendPathData.iStatus = 2) OR (stSuspendPathData.iStatus = 3) THEN
	stSuspendPathData.iStatus := 0;
END_IF

IF (bConnectedMethod AND NOT bBusyMethod) THEN
	IF (stSuspendPathData.iStatus = 0) THEN
	(* Setup method calling parameters *)
		(* Method identifier *)
		sObjectIDentifier := stSuspendPathData.sObjectID;
		sMethodIdentifier := stSuspendPathData.sMethodID;
	
		(* Method Inputs *)
		stSuspendPathData.stInput.iPath := nPathNo;
		(* Fill input data area with method arguments *)
		MEMSET(ADR(aInputData), 0 ,SIZEOF(aInputData));
		nOffset := 0;
		nOffset := nOffset + MEMCPY(ADR(aInputData)+nOffset, ADR(stSuspendPathData.stInput),	MIN(SIZEOF(stSuspendPathData.stInput), (SIZEOF(aInputData)-nOffset)) );
		(* Number of input arguments *)
		nNoOfInputArgs := stSuspendPathData.iNoOfInputArgs;
		(* Set up input argument information *)
		MEMSET(ADR(aInputArgInfo), 0, SIZEOF(aInputArgInfo));
		aInputArgInfo[1].DataType := eUAType_UInt16;
		aInputArgInfo[1].ValueRank := -1;	// -1: Scalar 
		aInputArgInfo[1].nLenData := SIZEOF(stSuspendPathData.stInput.iPath);
		
		(* Method outputs *)
		(* Clear output data area *)
		(* Number of output arguments *)
		nNoOfOutputArgs := stSuspendPathData.iNoOfOutputArgs;
		(* Set up output argument information *)
		MEMSET(ADR(aOutputArgInfo), 0, SIZEOF(aOutputArgInfo));
		aOutputArgInfo[1].DataType := eUAType_Uint16;
		aOutputArgInfo[1].ValueRank := -1;
		aOutputArgInfo[1].nLenData := SIZEOF(stSuspendPathData.stOutput.eStatus);
		aOutputArgInfo[2].DataType := eUAType_String;
		aOutputArgInfo[2].ValueRank := -1;
		aOutputArgInfo[2].nLenData := SIZEOF(stSuspendPathData.stOutput.sMessage);
		(* Set up output  *)
		MEMSET(ADR(stSuspendPathData.stOutput), 0, SIZEOF(stSuspendPathData.stOutput));
		stSuspendPathData.stOutput.nNumberOfOutputArguments := nNoOfOutputArgs;
		stSuspendPathData.stOutput.stOutputArgInfo[1] := aOutputArgInfo[1];
		stSuspendPathData.stOutput.stOutputArgInfo[2] := aOutputArgInfo[2];
	
		(* Execute FB *)
		fbCallMethod.nNumberOfInputArguments := nNoOfInputArgs;
		fbCallMethod.pInputArgInfo := ADR(aInputArgInfo);
		fbCallMethod.cbInputArgInfo := (SIZEOF(aInputArgInfo[1])*nNoOfInputArgs);
		fbCallMethod.pInputArgData := ADR(aInputData);
		fbCallMethod.cbInputArgData := nOffset;
		fbCallMethod.nNumberOfOutputArguments := nNoOfOutputArgs; 
		fbCallMethod.pOutputArgInfo := ADR(aOutputArgInfo); 
		fbCallMethod.cbOutputArgInfo := (SIZEOF(aOutputArgInfo[1]) * nNoOfOutputArgs); 
		fbCallMethod.pOutputArgInfoAndData := ADR(stSuspendPathData.stOutput);
		fbCallMethod.cbOutputArgInfoAndData := SIZEOF(stSuspendPathData.stOutput);
		
		stSuspendPathData.iStatus := 1;
		bCallMethod := TRUE;
		
	ELSIF (stSuspendPathData.iStatus = 1) THEN
		// Method call Completed...
		IF (eStateMethod = E_TrackClientState.Connected) THEN
			// Method call OK
			IF (stSuspendPathData.stOutput.eStatus = E_MMServerStatus.eMMServerStatus_Success) THEN
				// Method returned OK
				stSuspendPathData.iStatus := 2;
			ELSE
				// Method returned with error
				stSuspendPathData.iStatus := 3;
				stSuspendPathData.stOutput.sMessage;
			END_IF
		ELSIF (eStateMethod = E_TrackClientState.Error) THEN
			// Method call failed
			stSuspendPathData.iStatus := 3;
		END_IF
		
	END_IF
END_IF

M_CallSuspendPath := stSuspendPathData.iStatus;
END_METHOD

METHOD PROTECTED M_CallTrafficLightColor : INT
VAR_INPUT
END_VAR
IF (stTrafficLightColorData.iStatus = 2) OR (stTrafficLightColorData.iStatus = 3) THEN
	stTrafficLightColorData.iStatus := 0;
END_IF

IF (bConnectedMethod AND NOT bBusyMethod) THEN
	IF (stTrafficLightColorData.iStatus = 0) THEN
	(* Setup method calling parameters *)
		(* Method identifier *)
		sObjectIDentifier := stTrafficLightColorData.sObjectID;
		sMethodIdentifier := stTrafficLightColorData.sMethodID;
	
		(* Method Inputs *)
		stTrafficLightColorData.stInput.sCellID := sCellID;
		stTrafficLightColorData.stInput.sID := CONCAT(sCellID, '_TL');
		(* Fill input data area with method arguments *)
		MEMSET(ADR(aInputData), 0 ,SIZEOF(aInputData));
		nOffset := 0;
		nOffset := nOffset + MEMCPY(ADR(aInputData)+nOffset, ADR(stTrafficLightColorData.stInput),	MIN(SIZEOF(stTrafficLightColorData.stInput), (SIZEOF(aInputData)-nOffset)) );
		(* Number of input arguments *)
		nNoOfInputArgs := stTrafficLightColorData.iNoOfInputArgs;
		(* Set up input argument information *)
		MEMSET(ADR(aInputArgInfo), 0, SIZEOF(aInputArgInfo));
		aInputArgInfo[1].DataType := eUAType_String;
		aInputArgInfo[1].ValueRank := -1;	// -1: Scalar 
		aInputArgInfo[1].nLenData := SIZEOF(stTrafficLightColorData.stInput.sCellID);
		aInputArgInfo[2].DataType := eUAType_String;
		aInputArgInfo[2].ValueRank := -1;	// -1: Scalar 
		aInputArgInfo[2].nLenData := SIZEOF(stTrafficLightColorData.stInput.sID);
		
		(* Method outputs *)
		(* Clear output data area *)
		(* Number of output arguments *)
		nNoOfOutputArgs := stTrafficLightColorData.iNoOfOutputArgs;
		(* Set up output argument information *)
		MEMSET(ADR(aOutputArgInfo), 0, SIZEOF(aOutputArgInfo));
		aOutputArgInfo[1].DataType := eUAType_Uint16;
		aOutputArgInfo[1].ValueRank := -1;
		aOutputArgInfo[1].nLenData := SIZEOF(stTrafficLightColorData.stOutput.eStatus);
		aOutputArgInfo[2].DataType := eUAType_String;
		aOutputArgInfo[2].ValueRank := -1;
		aOutputArgInfo[2].nLenData := SIZEOF(stTrafficLightColorData.stOutput.sMessage);
		aOutputArgInfo[3].DataType := eUAType_Int16;
		aOutputArgInfo[3].ValueRank := -1;
		aOutputArgInfo[3].nLenData := SIZEOF(stTrafficLightColorData.stOutput.nTrafficLightColor);
		(* Set up output  *)
		MEMSET(ADR(stTrafficLightColorData.stOutput), 0, SIZEOF(stTrafficLightColorData.stOutput));
		stTrafficLightColorData.stOutput.nNumberOfOutputArguments := nNoOfOutputArgs;
		stTrafficLightColorData.stOutput.stOutputArgInfo[1] := aOutputArgInfo[1];
		stTrafficLightColorData.stOutput.stOutputArgInfo[2] := aOutputArgInfo[2];
		stTrafficLightColorData.stOutput.stOutputArgInfo[3] := aOutputArgInfo[3];
	
		(* Execute FB *)
		fbCallMethod.nNumberOfInputArguments := nNoOfInputArgs;
		fbCallMethod.pInputArgInfo := ADR(aInputArgInfo);
		fbCallMethod.cbInputArgInfo := (SIZEOF(aInputArgInfo[1])*nNoOfInputArgs);
		fbCallMethod.pInputArgData := ADR(aInputData);
		fbCallMethod.cbInputArgData := nOffset;
		fbCallMethod.nNumberOfOutputArguments := nNoOfOutputArgs; 
		fbCallMethod.pOutputArgInfo := ADR(aOutputArgInfo); 
		fbCallMethod.cbOutputArgInfo := (SIZEOF(aOutputArgInfo[1]) * nNoOfOutputArgs); 
		fbCallMethod.pOutputArgInfoAndData := ADR(stTrafficLightColorData.stOutput);
		fbCallMethod.cbOutputArgInfoAndData := SIZEOF(stTrafficLightColorData.stOutput);
		
		stTrafficLightColorData.iStatus := 1;
		bCallMethod := TRUE;
		
	ELSIF (stTrafficLightColorData.iStatus = 1) THEN
		// Method call Completed...
		IF (eStateMethod = E_TrackClientState.Connected) THEN
			// Method call OK
			IF (stTrafficLightColorData.stOutput.eStatus = E_MMServerStatus.eMMServerStatus_Success) THEN
				// Method returned OK
				stTrafficLightColorData.iStatus := 2;
			ELSE
				// Method returned with error
				stTrafficLightColorData.iStatus := 3;
				stTrafficLightColorData.stOutput.sMessage;
				stTrafficLightColorData.stOutput.nTrafficLightColor;
			END_IF
		ELSIF (eStateMethod = E_TrackClientState.Error) THEN
			// Method call failed
			stTrafficLightColorData.iStatus := 3;
		END_IF
		
	END_IF
END_IF

M_CallTrafficLightColor := stTrafficLightColorData.iStatus;
END_METHOD

METHOD PROTECTED M_CallUpdateStationBuffer : INT
VAR_INPUT
	sStationID			: STRING(30);
	eBufferType			: E_MMStationBuffer;
	nBufferIndex		: USINT;	
	nVehicleID			: UINT;
	sCarrierID			: STRING(30);
	nTicket				: UINT;
	nPriority			: UINT;
END_VAR
VAR
END_VAR
IF (stUpdateStationBufferData.iStatus = 2) OR (stUpdateStationBufferData.iStatus = 3) THEN
	stUpdateStationBufferData.iStatus := 0;
END_IF

IF (bConnectedMethod AND NOT bBusyMethod) THEN
	IF (stUpdateStationBufferData.iStatus = 0) THEN
	(* Setup method calling parameters *)
		(* Method identifier *)
		sObjectIDentifier := stUpdateStationBufferData.sObjectID;
		sMethodIdentifier := stUpdateStationBufferData.sMethodID;
	
		(* Method Inputs *)
		stUpdateStationBufferData.stInput.sStationID := sStationID;
		stUpdateStationBufferData.stInput.eStationBufferType := eBufferType;
		stUpdateStationBufferData.stInput.nIndex := nBufferIndex;
		stUpdateStationBufferData.stInput.nVehicleID := nVehicleID;
		stUpdateStationBufferData.stInput.sCarrierID := sCarrierID;
		stUpdateStationBufferData.stInput.nTicket := nTicket;
		stUpdateStationBufferData.stInput.nPriority := nPriority;
		
		(* Fill input data area with method arguments *)
		MEMSET(ADR(aInputData), 0 ,SIZEOF(aInputData));
		nOffset := 0;
		nOffset := nOffset + MEMCPY(ADR(aInputData)+nOffset, ADR(stUpdateStationBufferData.stInput),	MIN(SIZEOF(stUpdateStationBufferData.stInput), (SIZEOF(aInputData)-nOffset)) );
		(* Number of input arguments *)
		nNoOfInputArgs := stUpdateStationBufferData.iNoOfInputArgs;
		(* Set up input argument information *)
		MEMSET(ADR(aInputArgInfo), 0, SIZEOF(aInputArgInfo));
		aInputArgInfo[1].DataType := eUAType_String;
		aInputArgInfo[1].ValueRank := -1;	// -1: Scalar 
		aInputArgInfo[1].nLenData := SIZEOF(stUpdateStationBufferData.stInput.sStationID);
		aInputArgInfo[2].DataType := eUAType_UInt16;
		aInputArgInfo[2].ValueRank := -1;	// -1: Scalar 
		aInputArgInfo[2].nLenData := SIZEOF(stUpdateStationBufferData.stInput.eStationBufferType);
		aInputArgInfo[3].DataType := eUAType_Byte;
		aInputArgInfo[3].ValueRank := -1;	// -1: Scalar 
		aInputArgInfo[3].nLenData := SIZEOF(stUpdateStationBufferData.stInput.nIndex);
		aInputArgInfo[4].DataType := eUAType_UInt16;
		aInputArgInfo[4].ValueRank := -1;	// -1: Scalar 
		aInputArgInfo[4].nLenData := SIZEOF(stUpdateStationBufferData.stInput.nVehicleID);
		aInputArgInfo[5].DataType := eUAType_String;
		aInputArgInfo[5].ValueRank := -1;	// -1: Scalar 
		aInputArgInfo[5].nLenData := SIZEOF(stUpdateStationBufferData.stInput.sCarrierID);
		aInputArgInfo[6].DataType := eUAType_UInt16;
		aInputArgInfo[6].ValueRank := -1;	// -1: Scalar 
		aInputArgInfo[6].nLenData := SIZEOF(stUpdateStationBufferData.stInput.nTicket);
		aInputArgInfo[7].DataType := eUAType_UInt16;
		aInputArgInfo[7].ValueRank := -1;	// -1: Scalar 
		aInputArgInfo[7].nLenData := SIZEOF(stUpdateStationBufferData.stInput.nPriority);
		
		(* Method outputs *)
		(* Clear output data area *)
		(* Number of output arguments *)
		nNoOfOutputArgs := stUpdateStationBufferData.iNoOfOutputArgs;
		(* Set up output argument information *)
		MEMSET(ADR(aOutputArgInfo), 0, SIZEOF(aOutputArgInfo));
		aOutputArgInfo[1].DataType := eUAType_Uint16;
		aOutputArgInfo[1].ValueRank := -1;
		aOutputArgInfo[1].nLenData := SIZEOF(stUpdateStationBufferData.stOutput.eStatus);
		aOutputArgInfo[2].DataType := eUAType_String;
		aOutputArgInfo[2].ValueRank := -1;
		aOutputArgInfo[2].nLenData := SIZEOF(stUpdateStationBufferData.stOutput.sMessage);
		(* Set up output  *)
		MEMSET(ADR(stUpdateStationBufferData.stOutput), 0, SIZEOF(stUpdateStationBufferData.stOutput));
		stUpdateStationBufferData.stOutput.nNumberOfOutputArguments := nNoOfOutputArgs;
		stUpdateStationBufferData.stOutput.stOutputArgInfo[1] := aOutputArgInfo[1];
		stUpdateStationBufferData.stOutput.stOutputArgInfo[2] := aOutputArgInfo[2];
	
		(* Execute FB *)
		fbCallMethod.nNumberOfInputArguments := nNoOfInputArgs;
		fbCallMethod.pInputArgInfo := ADR(aInputArgInfo);
		fbCallMethod.cbInputArgInfo := (SIZEOF(aInputArgInfo[1])*nNoOfInputArgs);
		fbCallMethod.pInputArgData := ADR(aInputData);
		fbCallMethod.cbInputArgData := nOffset;
		fbCallMethod.nNumberOfOutputArguments := nNoOfOutputArgs; 
		fbCallMethod.pOutputArgInfo := ADR(aOutputArgInfo); 
		fbCallMethod.cbOutputArgInfo := (SIZEOF(aOutputArgInfo[1]) * nNoOfOutputArgs); 
		fbCallMethod.pOutputArgInfoAndData := ADR(stUpdateStationBufferData.stOutput);
		fbCallMethod.cbOutputArgInfoAndData := SIZEOF(stUpdateStationBufferData.stOutput);
		
		stUpdateStationBufferData.iStatus := 1;
		bCallMethod := TRUE;
		
	ELSIF (stUpdateStationBufferData.iStatus = 1) THEN
		// Method call Completed...
		IF (eStateMethod = E_TrackClientState.Connected) THEN
			// Method call OK
			IF (stUpdateStationBufferData.stOutput.eStatus = E_MMServerStatus.eMMServerStatus_Success) THEN
				// Method returned OK
				stUpdateStationBufferData.iStatus := 2;
			ELSE
				// Method returned with error
				stUpdateStationBufferData.iStatus := 3;
				stUpdateStationBufferData.stOutput.sMessage;
			END_IF
		ELSIF (eStateMethod = E_TrackClientState.Error) THEN
			// Method call failed
			stUpdateStationBufferData.iStatus := 3;
		END_IF
		
	END_IF
ELSE
	M_CallUpdateStationBuffer := -1;
	RETURN;
END_IF

M_CallUpdateStationBuffer := stUpdateStationBufferData.iStatus;
END_METHOD

METHOD M_CallUpdateVehicleMappingData : INT
VAR_INPUT
	nVehicleID			: UINT;										(* Magnemotion Vehicle ID *)
	sCarrierID			: STRING(30);								(* Carrier ID *)
	bTool				: BOOL;										(*  *)
	sToolID				: STRING(30);								(* Tool ID *)
	bMaterial			: BOOL;										(*  *)
	sMaterialID			: STRING(30);								(* Material ID string *)
END_VAR
VAR
END_VAR
IF (stUpdateVehicleMappingDataData.iStatus = 2) OR (stUpdateVehicleMappingDataData.iStatus = 3) THEN
	stUpdateVehicleMappingDataData.iStatus := 0;
END_IF

IF (bConnectedMethod AND NOT bBusyMethod) THEN
	IF (stUpdateVehicleMappingDataData.iStatus = 0) THEN
	(* Setup method calling parameters *)
		(* Method identifier *)
		sObjectIDentifier := stUpdateVehicleMappingDataData.sObjectID;
		sMethodIdentifier := stUpdateVehicleMappingDataData.sMethodID;
	
		(* Method Inputs *)
		stUpdateVehicleMappingDataData.stInput.nVehicleID := nVehicleID;
		stUpdateVehicleMappingDataData.stInput.sCarrierID := sCarrierID;
		stUpdateVehicleMappingDataData.stInput.bTool := bTool;
		stUpdateVehicleMappingDataData.stInput.sToolID := sToolID;
		stUpdateVehicleMappingDataData.stInput.bMaterial := bMaterial;
		stUpdateVehicleMappingDataData.stInput.sMaterialID := sMaterialID;
		
		(* Fill input data area with method arguments *)
		MEMSET(ADR(aInputData), 0 ,SIZEOF(aInputData));
		nOffset := 0;
		nOffset := nOffset + MEMCPY(ADR(aInputData)+nOffset, ADR(stUpdateVehicleMappingDataData.stInput),	MIN(SIZEOF(stUpdateVehicleMappingDataData.stInput), (SIZEOF(aInputData)-nOffset)) );
		(* Number of input arguments *)
		nNoOfInputArgs := stUpdateVehicleMappingDataData.iNoOfInputArgs;
		(* Set up input argument information *)
		MEMSET(ADR(aInputArgInfo), 0, SIZEOF(aInputArgInfo));
		aInputArgInfo[1].DataType := eUAType_UInt16;
		aInputArgInfo[1].ValueRank := -1;	// -1: Scalar 
		aInputArgInfo[1].nLenData := SIZEOF(stUpdateVehicleMappingDataData.stInput.nVehicleID);
		aInputArgInfo[2].DataType := eUAType_String;
		aInputArgInfo[2].ValueRank := -1;	// -1: Scalar 
		aInputArgInfo[2].nLenData := SIZEOF(stUpdateVehicleMappingDataData.stInput.sCarrierID);
		aInputArgInfo[3].DataType := eUAType_Boolean;
		aInputArgInfo[3].ValueRank := -1;	// -1: Scalar 
		aInputArgInfo[3].nLenData := SIZEOF(stUpdateVehicleMappingDataData.stInput.bTool);
		aInputArgInfo[4].DataType := eUAType_String;
		aInputArgInfo[4].ValueRank := -1;	// -1: Scalar 
		aInputArgInfo[4].nLenData := SIZEOF(stUpdateVehicleMappingDataData.stInput.sToolID);
		aInputArgInfo[5].DataType := eUAType_Boolean;
		aInputArgInfo[5].ValueRank := -1;	// -1: Scalar 
		aInputArgInfo[5].nLenData := SIZEOF(stUpdateVehicleMappingDataData.stInput.bMaterial);
		aInputArgInfo[6].DataType := eUAType_String;
		aInputArgInfo[6].ValueRank := -1;	// -1: Scalar 
		aInputArgInfo[6].nLenData := SIZEOF(stUpdateVehicleMappingDataData.stInput.sMaterialID);
		
		(* Method outputs *)
		(* Clear output data area *)
		(* Number of output arguments *)
		nNoOfOutputArgs := stUpdateVehicleMappingDataData.iNoOfOutputArgs;
		(* Set up output argument information *)
		MEMSET(ADR(aOutputArgInfo), 0, SIZEOF(aOutputArgInfo));
		aOutputArgInfo[1].DataType := eUAType_Uint16;
		aOutputArgInfo[1].ValueRank := -1;
		aOutputArgInfo[1].nLenData := SIZEOF(stUpdateVehicleMappingDataData.stOutput.eStatus);
		aOutputArgInfo[2].DataType := eUAType_String;
		aOutputArgInfo[2].ValueRank := -1;
		aOutputArgInfo[2].nLenData := SIZEOF(stUpdateVehicleMappingDataData.stOutput.sMessage);
		(* Set up output  *)
		MEMSET(ADR(stUpdateVehicleMappingDataData.stOutput), 0, SIZEOF(stUpdateVehicleMappingDataData.stOutput));
		stUpdateVehicleMappingDataData.stOutput.nNumberOfOutputArguments := nNoOfOutputArgs;
		stUpdateVehicleMappingDataData.stOutput.stOutputArgInfo[1] := aOutputArgInfo[1];
		stUpdateVehicleMappingDataData.stOutput.stOutputArgInfo[2] := aOutputArgInfo[2];
	
		(* Execute FB *)
		fbCallMethod.nNumberOfInputArguments := nNoOfInputArgs;
		fbCallMethod.pInputArgInfo := ADR(aInputArgInfo);
		fbCallMethod.cbInputArgInfo := (SIZEOF(aInputArgInfo[1])*nNoOfInputArgs);
		fbCallMethod.pInputArgData := ADR(aInputData);
		fbCallMethod.cbInputArgData := nOffset;
		fbCallMethod.nNumberOfOutputArguments := nNoOfOutputArgs; 
		fbCallMethod.pOutputArgInfo := ADR(aOutputArgInfo); 
		fbCallMethod.cbOutputArgInfo := (SIZEOF(aOutputArgInfo[1]) * nNoOfOutputArgs); 
		fbCallMethod.pOutputArgInfoAndData := ADR(stUpdateVehicleMappingDataData.stOutput);
		fbCallMethod.cbOutputArgInfoAndData := SIZEOF(stUpdateVehicleMappingDataData.stOutput);
		
		stUpdateVehicleMappingDataData.iStatus := 1;
		bCallMethod := TRUE;
		
	ELSIF (stUpdateVehicleMappingDataData.iStatus = 1) THEN
		// Method call Completed...
		IF (eStateMethod = E_TrackClientState.Connected) THEN
			// Method call OK
			IF (stUpdateVehicleMappingDataData.stOutput.eStatus = E_MMServerStatus.eMMServerStatus_Success) THEN
				// Method returned OK
				stUpdateVehicleMappingDataData.iStatus := 2;
				// Trig vehicle data reading because data has changed
				M_VehicleToReadAdd(stUpdateVehicleMappingDataData.stInput.nVehicleID);
				
			ELSE
				// Method returned with error
				stUpdateVehicleMappingDataData.iStatus := 3;
				stUpdateVehicleMappingDataData.stOutput.sMessage;
				
			END_IF
			
		ELSIF (eStateMethod = E_TrackClientState.Error) THEN
			// Method call failed
			stUpdateVehicleMappingDataData.iStatus := 3;
			
		END_IF
		
	END_IF
ELSE
	M_CallUpdateVehicleMappingData := -1;
	RETURN;
	
END_IF

M_CallUpdateVehicleMappingData := stUpdateVehicleMappingDataData.iStatus;
END_METHOD

METHOD M_CallUpdateVehicleMontage : INT
VAR_INPUT
	nVehicleID			: UINT;										(* Magnemotion Vehicle ID *)
	bTool				: BOOL;										(*  *)
	sToolID				: STRING(30);								(* Tool ID *)
	bMaterial			: BOOL;										(*  *)
	sMaterialID			: STRING(30);								(* Material ID string *)
	bReserved			: BOOL;										(* TRUE signals vehicle is reserved for montage line *)
END_VAR
VAR
END_VAR
IF (stUpdateVehicleMontageData.iStatus = 2) OR (stUpdateVehicleMontageData.iStatus = 3) THEN
	stUpdateVehicleMontageData.iStatus := 0;
END_IF

IF (bConnectedMethod AND NOT bBusyMethod) THEN
	IF (stUpdateVehicleMontageData.iStatus = 0) THEN
	(* Setup method calling parameters *)
		(* Method identifier *)
		sObjectIDentifier := stUpdateVehicleMontageData.sObjectID;
		sMethodIdentifier := stUpdateVehicleMontageData.sMethodID;
	
		(* Method Inputs *)
		stUpdateVehicleMontageData.stInput.eInputType := E_MMVehicleInputType.eMMVehicleInputType_VehicleID;
		stUpdateVehicleMontageData.stInput.sInput := UINT_TO_STRING(nVehicleID);
		stUpdateVehicleMontageData.stInput.bTool := bTool;
		stUpdateVehicleMontageData.stInput.sToolID := sToolID;
		stUpdateVehicleMontageData.stInput.bMaterial := bMaterial;
		stUpdateVehicleMontageData.stInput.sMaterialID := sMaterialID;
		stUpdateVehicleMontageData.stInput.bReserved := bReserved;
		
		(* Fill input data area with method arguments *)
		MEMSET(ADR(aInputData), 0 ,SIZEOF(aInputData));
		nOffset := 0;
		nOffset := nOffset + MEMCPY(ADR(aInputData)+nOffset, ADR(stUpdateVehicleMontageData.stInput),	MIN(SIZEOF(stUpdateVehicleMontageData.stInput), (SIZEOF(aInputData)-nOffset)) );
		(* Number of input arguments *)
		nNoOfInputArgs := stUpdateVehicleMontageData.iNoOfInputArgs;
		(* Set up input argument information *)
		MEMSET(ADR(aInputArgInfo), 0, SIZEOF(aInputArgInfo));
		aInputArgInfo[1].DataType := eUAType_UInt16;
		aInputArgInfo[1].ValueRank := -1;	// -1: Scalar 
		aInputArgInfo[1].nLenData := SIZEOF(stUpdateVehicleMontageData.stInput.eInputType);
		aInputArgInfo[2].DataType := eUAType_String;
		aInputArgInfo[2].ValueRank := -1;	// -1: Scalar 
		aInputArgInfo[2].nLenData := SIZEOF(stUpdateVehicleMontageData.stInput.sInput);
		aInputArgInfo[3].DataType := eUAType_Boolean;
		aInputArgInfo[3].ValueRank := -1;	// -1: Scalar 
		aInputArgInfo[3].nLenData := SIZEOF(stUpdateVehicleMontageData.stInput.bTool);
		aInputArgInfo[4].DataType := eUAType_String;
		aInputArgInfo[4].ValueRank := -1;	// -1: Scalar 
		aInputArgInfo[4].nLenData := SIZEOF(stUpdateVehicleMontageData.stInput.sToolID);
		aInputArgInfo[5].DataType := eUAType_Boolean;
		aInputArgInfo[5].ValueRank := -1;	// -1: Scalar 
		aInputArgInfo[5].nLenData := SIZEOF(stUpdateVehicleMontageData.stInput.bMaterial);
		aInputArgInfo[6].DataType := eUAType_String;
		aInputArgInfo[6].ValueRank := -1;	// -1: Scalar 
		aInputArgInfo[6].nLenData := SIZEOF(stUpdateVehicleMontageData.stInput.sMaterialID);
		aInputArgInfo[7].DataType := eUAType_Boolean;
		aInputArgInfo[7].ValueRank := -1;	// -1: Scalar 
		aInputArgInfo[7].nLenData := SIZEOF(stUpdateVehicleMontageData.stInput.bReserved);
		
		(* Method outputs *)
		(* Clear output data area *)
		(* Number of output arguments *)
		nNoOfOutputArgs := stUpdateVehicleMontageData.iNoOfOutputArgs;
		(* Set up output argument information *)
		MEMSET(ADR(aOutputArgInfo), 0, SIZEOF(aOutputArgInfo));
		aOutputArgInfo[1].DataType := eUAType_Uint16;
		aOutputArgInfo[1].ValueRank := -1;
		aOutputArgInfo[1].nLenData := SIZEOF(stUpdateVehicleMontageData.stOutput.eStatus);
		aOutputArgInfo[2].DataType := eUAType_String;
		aOutputArgInfo[2].ValueRank := -1;
		aOutputArgInfo[2].nLenData := SIZEOF(stUpdateVehicleMontageData.stOutput.sMessage);
		(* Set up output  *)
		MEMSET(ADR(stUpdateVehicleMontageData.stOutput), 0, SIZEOF(stUpdateVehicleMontageData.stOutput));
		stUpdateVehicleMontageData.stOutput.nNumberOfOutputArguments := nNoOfOutputArgs;
		stUpdateVehicleMontageData.stOutput.stOutputArgInfo[1] := aOutputArgInfo[1];
		stUpdateVehicleMontageData.stOutput.stOutputArgInfo[2] := aOutputArgInfo[2];
	
		(* Execute FB *)
		fbCallMethod.nNumberOfInputArguments := nNoOfInputArgs;
		fbCallMethod.pInputArgInfo := ADR(aInputArgInfo);
		fbCallMethod.cbInputArgInfo := (SIZEOF(aInputArgInfo[1])*nNoOfInputArgs);
		fbCallMethod.pInputArgData := ADR(aInputData);
		fbCallMethod.cbInputArgData := nOffset;
		fbCallMethod.nNumberOfOutputArguments := nNoOfOutputArgs; 
		fbCallMethod.pOutputArgInfo := ADR(aOutputArgInfo); 
		fbCallMethod.cbOutputArgInfo := (SIZEOF(aOutputArgInfo[1]) * nNoOfOutputArgs); 
		fbCallMethod.pOutputArgInfoAndData := ADR(stUpdateVehicleMontageData.stOutput);
		fbCallMethod.cbOutputArgInfoAndData := SIZEOF(stUpdateVehicleMontageData.stOutput);
		
		stUpdateVehicleMontageData.iStatus := 1;
		bCallMethod := TRUE;
		
	ELSIF (stUpdateVehicleMontageData.iStatus = 1) THEN
		// Method call Completed...
		IF (UINT_TO_STRING(nVehicleID) = stUpdateVehicleMontageData.stInput.sInput) THEN
			IF (eStateMethod = E_TrackClientState.Connected) THEN
				// Method call OK
				IF (stUpdateVehicleMontageData.stOutput.eStatus = E_MMServerStatus.eMMServerStatus_Success) THEN
					// Method returned OK
					stUpdateVehicleMontageData.iStatus := 2;
					// Trig vehicle data reading because data has changed
					M_VehicleToReadAdd(nVehicleID);
									
				ELSE
					// Method returned with error
					stUpdateVehicleMontageData.iStatus := 3;
					stUpdateVehicleMontageData.stOutput.sMessage;
					
				END_IF
				
			ELSIF (eStateMethod = E_TrackClientState.Error) THEN
				// Method call failed
				stUpdateVehicleMontageData.iStatus := 3;
	
			END_IF
		ELSE
			// Wrong vehicle ID
			F_LogLine('TC_VMD: Wrong Vehicle ID (%d)', nVehicleID);
			
		END_IF
	END_IF
ELSE
	M_CallUpdateVehicleMontage := -1;
	RETURN;

END_IF

M_CallUpdateVehicleMontage := stUpdateVehicleMontageData.iStatus;
END_METHOD

METHOD PROTECTED M_CallUpdateVehicleOwner : INT
VAR_INPUT
	nVehicleID			: UINT;										(* Magnemotion Vehicle ID *)
	eInputType			: E_MMVehicleInputType;
	sInput				: STRING(30);
	sCellID				: STRING(30);
END_VAR
VAR
END_VAR
IF (stUpdateVehicleOwnerData.iStatus = 2) OR (stUpdateVehicleOwnerData.iStatus = 3) THEN
	stUpdateVehicleOwnerData.iStatus := 0;
END_IF

IF (bConnectedMethod AND NOT bBusyMethod) THEN
	IF (stUpdateVehicleOwnerData.iStatus = 0) THEN
	(* Setup method calling parameters *)
		(* Method identifier *)
		sObjectIDentifier := stUpdateVehicleOwnerData.sObjectID;
		sMethodIdentifier := stUpdateVehicleOwnerData.sMethodID;
	
		(* Method Inputs *)
		stUpdateVehicleOwnerData.stInput.eInputType := eInputType;
		stUpdateVehicleOwnerData.stInput.sInput := sInput;
		stUpdateVehicleOwnerData.stInput.sCellID := sCellID;
		
		(* Fill input data area with method arguments *)
		MEMSET(ADR(aInputData), 0 ,SIZEOF(aInputData));
		nOffset := 0;
		nOffset := nOffset + MEMCPY(ADR(aInputData)+nOffset, ADR(stUpdateVehicleOwnerData.stInput),	MIN(SIZEOF(stUpdateVehicleOwnerData.stInput), (SIZEOF(aInputData)-nOffset)) );
		(* Number of input arguments *)
		nNoOfInputArgs := stUpdateVehicleOwnerData.iNoOfInputArgs;
		(* Set up input argument information *)
		MEMSET(ADR(aInputArgInfo), 0, SIZEOF(aInputArgInfo));
		aInputArgInfo[1].DataType := eUAType_UInt16;
		aInputArgInfo[1].ValueRank := -1;	// -1: Scalar 
		aInputArgInfo[1].nLenData := SIZEOF(stUpdateVehicleOwnerData.stInput.eInputType);
		aInputArgInfo[2].DataType := eUAType_String;
		aInputArgInfo[2].ValueRank := -1;	// -1: Scalar 
		aInputArgInfo[2].nLenData := SIZEOF(stUpdateVehicleOwnerData.stInput.sInput);
		aInputArgInfo[3].DataType := eUAType_String;
		aInputArgInfo[3].ValueRank := -1;	// -1: Scalar 
		aInputArgInfo[3].nLenData := SIZEOF(stUpdateVehicleOwnerData.stInput.sCellID);
		
		(* Method outputs *)
		(* Clear output data area *)
		(* Number of output arguments *)
		nNoOfOutputArgs := stUpdateVehicleOwnerData.iNoOfOutputArgs;
		(* Set up output argument information *)
		MEMSET(ADR(aOutputArgInfo), 0, SIZEOF(aOutputArgInfo));
		aOutputArgInfo[1].DataType := eUAType_Uint16;
		aOutputArgInfo[1].ValueRank := -1;
		aOutputArgInfo[1].nLenData := SIZEOF(stUpdateVehicleOwnerData.stOutput.eStatus);
		aOutputArgInfo[2].DataType := eUAType_String;
		aOutputArgInfo[2].ValueRank := -1;
		aOutputArgInfo[2].nLenData := SIZEOF(stUpdateVehicleOwnerData.stOutput.sMessage);
		(* Set up output  *)
		MEMSET(ADR(stUpdateVehicleOwnerData.stOutput), 0, SIZEOF(stUpdateVehicleOwnerData.stOutput));
		stUpdateVehicleOwnerData.stOutput.nNumberOfOutputArguments := nNoOfOutputArgs;
		stUpdateVehicleOwnerData.stOutput.stOutputArgInfo[1] := aOutputArgInfo[1];
		stUpdateVehicleOwnerData.stOutput.stOutputArgInfo[2] := aOutputArgInfo[2];
	
		(* Execute FB *)
		fbCallMethod.nNumberOfInputArguments := nNoOfInputArgs;
		fbCallMethod.pInputArgInfo := ADR(aInputArgInfo);
		fbCallMethod.cbInputArgInfo := (SIZEOF(aInputArgInfo[1])*nNoOfInputArgs);
		fbCallMethod.pInputArgData := ADR(aInputData);
		fbCallMethod.cbInputArgData := nOffset;
		fbCallMethod.nNumberOfOutputArguments := nNoOfOutputArgs; 
		fbCallMethod.pOutputArgInfo := ADR(aOutputArgInfo); 
		fbCallMethod.cbOutputArgInfo := (SIZEOF(aOutputArgInfo[1]) * nNoOfOutputArgs); 
		fbCallMethod.pOutputArgInfoAndData := ADR(stUpdateVehicleOwnerData.stOutput);
		fbCallMethod.cbOutputArgInfoAndData := SIZEOF(stUpdateVehicleOwnerData.stOutput);
		
		stUpdateVehicleOwnerData.iStatus := 1;
		bCallMethod := TRUE;
		
	ELSIF (stUpdateVehicleOwnerData.iStatus = 1) THEN
		// Method call Completed...
		IF (eStateMethod = E_TrackClientState.Connected) THEN
			// Method call OK
			IF (stUpdateVehicleOwnerData.stOutput.eStatus = E_MMServerStatus.eMMServerStatus_Success) THEN
				// Method returned OK
				stUpdateVehicleOwnerData.iStatus := 2;
				// Trig vehicle data reading because data has changed
				M_VehicleToReadAdd(nVehicleID);
				
			ELSE
				// Method returned with error
				stUpdateVehicleOwnerData.iStatus := 3;
				stUpdateVehicleOwnerData.stOutput.sMessage;

			END_IF
		ELSIF (eStateMethod = E_TrackClientState.Error) THEN
			// Method call failed
			stUpdateVehicleOwnerData.iStatus := 3;

		END_IF
		
	END_IF
ELSE
	M_CallUpdateVehicleOwner := -1;
	RETURN;

END_IF

M_CallUpdateVehicleOwner := stUpdateVehicleOwnerData.iStatus;
END_METHOD

METHOD M_CallUpdateVehicleReservationData : INT
VAR_INPUT
	nVehicleID			: UINT;										(* Magnemotion vehicle ID *)
	sTargetStationID	: STRING(30);								(* Target station ID *)
	sCarrierID			: STRING(30);								(* Carrier ID *)
	sJobID				: STRING(30);								(* Job ID string *)
	nTicket				: UINT;										(* Ticket number *)
	nCarriersInPackage	: UINT;										(* Ticket size *)
	nPriority			: UINT;										(* Ticket priority *)
END_VAR
VAR
END_VAR
IF (stUpdateVehicleReservationDataData.iStatus = 2) OR (stUpdateVehicleReservationDataData.iStatus = 3) THEN
	stUpdateVehicleReservationDataData.iStatus := 0;
END_IF

IF (bConnectedMethod AND NOT bBusyMethod) THEN
	IF (stUpdateVehicleReservationDataData.iStatus = 0) THEN
	(* Setup method calling parameters *)
		(* Method identifier *)
		sObjectIDentifier := stUpdateVehicleReservationDataData.sObjectID;
		sMethodIdentifier := stUpdateVehicleReservationDataData.sMethodID;
	
		(* Method Inputs *)
		stUpdateVehicleReservationDataData.stInput.sTargetStationID := sTargetStationID;
		stUpdateVehicleReservationDataData.stInput.sCarrierID := sCarrierID;
		stUpdateVehicleReservationDataData.stInput.sJobID := sJobID;
		stUpdateVehicleReservationDataData.stInput.nTicket := nTicket;
		stUpdateVehicleReservationDataData.stInput.nCarriersInPackage := nCarriersInPackage;
		stUpdateVehicleReservationDataData.stInput.nPriority := nPriority;
		
		(* Fill input data area with method arguments *)
		MEMSET(ADR(aInputData), 0 ,SIZEOF(aInputData));
		nOffset := 0;
		nOffset := nOffset + MEMCPY(ADR(aInputData)+nOffset, ADR(stUpdateVehicleReservationDataData.stInput),	MIN(SIZEOF(stUpdateVehicleReservationDataData.stInput), (SIZEOF(aInputData)-nOffset)) );
		(* Number of input arguments *)
		nNoOfInputArgs := stUpdateVehicleReservationDataData.iNoOfInputArgs;
		(* Set up input argument information *)
		MEMSET(ADR(aInputArgInfo), 0, SIZEOF(aInputArgInfo));
		aInputArgInfo[1].DataType := eUAType_String;
		aInputArgInfo[1].ValueRank := -1;	// -1: Scalar 
		aInputArgInfo[1].nLenData := SIZEOF(stUpdateVehicleReservationDataData.stInput.sTargetStationID);
		aInputArgInfo[2].DataType := eUAType_String;
		aInputArgInfo[2].ValueRank := -1;	// -1: Scalar 
		aInputArgInfo[2].nLenData := SIZEOF(stUpdateVehicleReservationDataData.stInput.sCarrierID);
		aInputArgInfo[3].DataType := eUAType_String;
		aInputArgInfo[3].ValueRank := -1;	// -1: Scalar 
		aInputArgInfo[3].nLenData := SIZEOF(stUpdateVehicleReservationDataData.stInput.sJobID);
		aInputArgInfo[4].DataType := eUAType_UInt16;
		aInputArgInfo[4].ValueRank := -1;	// -1: Scalar 
		aInputArgInfo[4].nLenData := SIZEOF(stUpdateVehicleReservationDataData.stInput.nTicket);
		aInputArgInfo[5].DataType := eUAType_UInt16;
		aInputArgInfo[5].ValueRank := -1;	// -1: Scalar 
		aInputArgInfo[5].nLenData := SIZEOF(stUpdateVehicleReservationDataData.stInput.nCarriersInPackage);
		aInputArgInfo[6].DataType := eUAType_UInt16;
		aInputArgInfo[6].ValueRank := -1;	// -1: Scalar 
		aInputArgInfo[6].nLenData := SIZEOF(stUpdateVehicleReservationDataData.stInput.nPriority);
		
		(* Method outputs *)
		(* Clear output data area *)
		(* Number of output arguments *)
		nNoOfOutputArgs := stUpdateVehicleReservationDataData.iNoOfOutputArgs;
		(* Set up output argument information *)
		MEMSET(ADR(aOutputArgInfo), 0, SIZEOF(aOutputArgInfo));
		aOutputArgInfo[1].DataType := eUAType_Uint16;
		aOutputArgInfo[1].ValueRank := -1;
		aOutputArgInfo[1].nLenData := SIZEOF(stUpdateVehicleReservationDataData.stOutput.eStatus);
		aOutputArgInfo[2].DataType := eUAType_String;
		aOutputArgInfo[2].ValueRank := -1;
		aOutputArgInfo[2].nLenData := SIZEOF(stUpdateVehicleReservationDataData.stOutput.sMessage);
		(* Set up output  *)
		MEMSET(ADR(stUpdateVehicleReservationDataData.stOutput), 0, SIZEOF(stUpdateVehicleReservationDataData.stOutput));
		stUpdateVehicleReservationDataData.stOutput.nNumberOfOutputArguments := nNoOfOutputArgs;
		stUpdateVehicleReservationDataData.stOutput.stOutputArgInfo[1] := aOutputArgInfo[1];
		stUpdateVehicleReservationDataData.stOutput.stOutputArgInfo[2] := aOutputArgInfo[2];
	
